// ---- Library/10_Machine/18_HMI_Handshake/OLD_DUTs/E_PullOutConveyorCommandType.TcDUT
{attribute 'qualified_only'}
{attribute 'strict'}
TYPE
    E_PullOutConveyorCommandType :
    (
		SideA_FeedIn := 1, // Pull out conveyor A-side feed in box.
		SideB_FeedIn , // Pull out conveyor B-Side feed in box.
		Both_FeedIn, // Pull out conveyor both side feed in box.
		SideA_FeedOut, // Pull out conveyor A-side feed out box.
		SideB_FeedOut, // Pull out conveyor B-Side feed out box.
		Both_FeedOut, // Pull out conveyor both side feed out box.
        MoveForward, // Pull out conveyor motor move forward.
        MoveBackward, // Pull out conveyor motor move backward.
		SlideA_FeedOut_Ext, // Pullout Conveyor A-side feed out box, fast flow(Design by Johnson)
		SlideB_FeedOut_Ext, // Pullout Conveyor B-Side feed out box, fast flow(Design by Johnson)
		SlideA_FeedIn_Ext, // Pullout Conveyor A-side feed in box, fast flow(Design by Johnson)
		SlideB_FeedIn_Ext // Pullout Conveyor B-side feed in box, fast flow(Design by Johnson)
    );
END_TYPE

// ---- Library/10_Machine/18_HMI_Handshake/OLD_DUTs/E_PullOutConveyorState.TcDUT
{attribute 'qualified_only'}
{attribute 'strict'}
TYPE E_PullOutConveyorState :
(
	idle := 0,
	AutoMode,
	Free
);
END_TYPE

// ---- Library/10_Machine/18_HMI_Handshake/OLD_DUTs/E_RackState.TcDUT
{attribute 'qualified_only'}
{attribute 'strict'}
TYPE E_RackState :
(
	idle := 0,
	AddBoxes,
	ManualCtrl,
	FeedBox,
	Free,
	TransitingFeedBox,
	TransitingFree
);
END_TYPE

// ---- Library/10_Machine/18_HMI_Handshake/OLD_DUTs/E_ReloadRoundBelt_PickupArea.TcDUT
{attribute 'qualified_only'}
{attribute 'strict'}
TYPE
    E_ReloadRoundBelt_PickupArea :
    (
        Undefined := 0,
        WareHouseA := 1,
        WareHouseB := 2
        )UINT;
END_TYPE

// ---- Library/10_Machine/18_HMI_Handshake/OLD_DUTs/E_ReloadRoundBelt_PlaceAddress.TcDUT
{attribute 'qualified_only'}
{attribute 'strict'}
TYPE E_ReloadRoundBelt_PlaceAddress :
(
	Undefined := 0,
	A1,
	A2,
	A3,
	A4
);
END_TYPE

// ---- Library/10_Machine/18_HMI_Handshake/OLD_DUTs/E_ReloadRoundBelt_PlaceArea.TcDUT
{attribute 'qualified_only'}
{attribute 'strict'}
TYPE E_ReloadRoundBelt_PlaceArea :
(
	Undefined := 0,
	RoundBelt
)UINT;
END_TYPE

// ---- Library/10_Machine/18_HMI_Handshake/OLD_DUTs/E_RobotArea.TcDUT
{attribute 'qualified_only'}
{attribute 'strict'}
(* This enum is use to define Fanuc robot target position in the StorageArea,
In the StorageArea, areas excluding the Warehouse.
*)
TYPE
    E_RobotArea :
    (
        Undefined := 0,
        // 圓帶,B區
        RoundBelt := 1,
        // 緩衝區,C區
        BufferArea := 2,
        // 補料軌道,D區
        TransmitCV := 3,
//        // 簡易配針區,E區
//        SimpleAllocate := 4,
        // 入出料軌道,F區 (倉儲區軌道)
        InOutConveyor := 5,
//        // 倉儲預備區,G區
//        WareHouseA_Buffer := 6,
        // 回拔輸送帶,H區
        PullOutConveyor := 7,
        // 小手臂左 (操作面)
        ShippingRobotLeft := 8,
        // 小手臂右 (操作面)
        ShippingRobotRight := 9,
		// Shipping Store,K
		TransmitCV_End :=10,
		// Shipping Buffer , K
		ShippingBufferArea := 11,
		// 小手臂CCD Pos
		ShippingCCDPos	:= 12,
		// 小手臂 拔針排空盒
		ShippingFeedOutEmptyBox := 13
    );
END_TYPE

// ---- Library/10_Machine/18_HMI_Handshake/OLD_DUTs/E_RobotClamp.TcDUT
{attribute 'qualified_only'}
{attribute 'strict'}
TYPE E_RobotClamp :
(
	ClampA := 1,
	ClampB
);
END_TYPE

// ---- Library/10_Machine/18_HMI_Handshake/OLD_DUTs/E_RoundBeltStation.TcDUT
{attribute 'qualified_only'}
TYPE E_RoundBeltStation :
(
	Undefined := 0,
	Station01,
	Station02,
	Station03,
	Station04,
	Station05,
	Station06,
	Station07,
	Station08,
	Station09,
	Station10,
	Station11,
	Station12,
	Station13,
	Station14,
	Station15,
	Station16,
	Station17,
	Station18,
	Station19,
	Station20,
	Station21,
	Station22,
	Station23,
	Station24,
	Station25,
	Station26,
	Station27,
	Station28,
	Station29,
	Station30,
	Station31,
	Station32,
	Station33,
	Station34,
	Station35,
	Station36,
	Station37,
	Station38,
	Station39,
	Station40
)UINT;
END_TYPE

// ---- Library/10_Machine/18_HMI_Handshake/OLD_DUTs/E_SimpleAllocateTable.TcDUT
{attribute 'qualified_only'}
{attribute 'strict'}
TYPE E_SimpleAllocateTable :
(
    Box1 :=1,
    Box2,
    Box3,
    Box4
);
END_TYPE

// ---- Library/10_Machine/18_HMI_Handshake/OLD_DUTs/E_WareHouse.TcDUT
TYPE E_WareHouse :
(
	None := 0,
	WareHouseA := 1,
	WareHouseB := 2
);
END_TYPE

// ---- Library/10_Machine/18_HMI_Handshake/OLD_DUTs/E_WareHouseLayer.TcDUT
TYPE E_WareHouseLayer :
(
	Undefine := 0,
	Layer01 := 1,
	Layer02,
	Layer03,
	Layer04,
	Layer05,
	Layer06,
	Layer07,
	Layer08,
	Layer09,
	Layer10
);
END_TYPE

// ---- Library/10_Machine/18_HMI_Handshake/OLD_DUTs/E_WareHouseSlide.TcDUT
TYPE
    E_WareHouseSlide :
    (
        Undefine := 0,
        Slide01 := 1,
        Slide02,
        Slide03,
        Slide04,
        Slide05,
        Slide06,
        Slide07,
        Slide08,
        Slide09,
        Slide10,
        Slide11,
        Slide12,
        Slide13,
        Slide14,
        Slide15,
        Slide16,
        Slide17,
        Slide18,
        Slide19,
        Slide20
    );
END_TYPE

// ---- Library/10_Machine/18_HMI_Handshake/OLD_DUTs/stPositionCommand.TcDUT
TYPE
    stPositionCommand :
    STRUCT
        Xaxis_Pos : LREAL; // Robot X-axis position command
        Yaxis_Pos : LREAL; // Robot Y-axis position command
        Raxis_Pos : LREAL; // Robot R-axis Position command
    END_STRUCT
END_TYPE

// ---- Library/10_Machine/18_HMI_Handshake/OLD_DUTs/st_ads_AllocateMoveStructure.TcDUT
TYPE
    st_ads_AllocateMoveStructure :
    STRUCT
        //手臂夾爪 ex 0=>A爪 1=>B爪 and so on...	
        Clip         : LREAL;
        Frombox      : LREAL;
        Tobox        : LREAL;
        FromPosition : LREAL;
        ToPosition   : LREAL;
        HandShake    : st_HandshakeBase;
    END_STRUCT
END_TYPE

// ---- Library/10_Machine/18_HMI_Handshake/OLD_DUTs/st_ads_MachineReset.TcDUT
TYPE st_ads_MachineReset :
    STRUCT
        //清除各分區除了伺服軸外的所有動件(氣壓缸、馬達)的邏輯層錯誤
        ResetStorage    :BOOL;
        ResetAllocation :BOOL;
        ResetFGA        :BOOL;
        AllReset        :BOOL;// Machine reset signal, True: machine try to clear alarm and reset method 
    END_STRUCT
END_TYPE

// ---- Library/10_Machine/18_HMI_Handshake/OLD_DUTs/st_ads_OneAxisMoveWithoutPosition.TcDUT
TYPE st_ads_OneAxisMoveWithoutPosition :
STRUCT
	//Excute:BOOL;
	//Done:BOOL;
	//Busy  : BOOL;
	//Occupied : BOOL;
	
	HandShake					: st_HandshakeBase;
END_STRUCT
END_TYPE

// ---- Library/10_Machine/18_HMI_Handshake/OLD_DUTs/st_ads_OneAxisMoveWithPosition.TcDUT
TYPE st_ads_OneAxisMoveWithPosition :
STRUCT
	Clip:LREAL;
	Position:LREAL; 
	
	HandShake					: st_HandshakeBase;
END_STRUCT
END_TYPE

// ---- Library/10_Machine/18_HMI_Handshake/OLD_DUTs/st_ads_OutRobtToPlateMove.TcDUT
TYPE st_ads_OutRobtToPlateMove :
STRUCT
	//軌道 散針軌道 or 同尺寸軌道
Slide :LREAL;
Clip:LREAL;
//鐵盤位置
PlatePosition :LREAL;
//Excute :bool;
//Done    :BOOL;
HandShake					: st_HandshakeBase;
END_STRUCT
END_TYPE

// ---- Library/10_Machine/18_HMI_Handshake/OLD_DUTs/st_ads_RobotToAllocateMove.TcDUT
TYPE
    st_ads_RobotToAllocateMove :
    STRUCT
        //圓帶位置
        AllocatePosition : LREAL;
        //手臂夾爪 ex 0=>A爪 1=>B爪
        RobotClip : LREAL;
        //倉儲區域 ex>A,B
        Area : LREAL;
        //倉儲層
        WarehouseLayer : LREAL;
        //倉儲道
        WarehouseOrbit : LREAL;
        // :BOOL;
        //Done :BOOL;
        HandShake : st_HandshakeBase;
    END_STRUCT
END_TYPE

// ---- Library/10_Machine/18_HMI_Handshake/OLD_DUTs/ST_Alarm_Tmax.TcDUT
TYPE ST_Alarm_Tmax :
STRUCT
		Trigger		:BOOL; //	Alarm trigger point
		ID			: UDINT; //	Alarm ID
		Value		: DINT; //	Alarm Value
		Message		: T_MaxString; //	Alarm Message
		Category	: DINT; //	Alarm Category
		DateTime	: ARRAY[0..6] OF DINT;
		ackDateTime : ARRAY[0..6] OF DINT;
END_STRUCT
END_TYPE

// ---- Library/10_Machine/18_HMI_Handshake/OLD_DUTs/st_AllocateCircleMoveStructure.TcDUT
TYPE st_AllocateCircleMoveStructure :
STRUCT
	Latch : LREAL;
	Position :LREAL;
//	Excute	:BOOL;
//	Done	 :BOOL;
//	Busy  : BOOL;
//	Occupied : BOOL;	
	HandShake					: st_HandshakeBase;
END_STRUCT
END_TYPE

// ---- Library/10_Machine/18_HMI_Handshake/OLD_DUTs/st_AllocateRobotNeedlingMove.TcDUT
TYPE st_AllocateRobotNeedlingMove :
STRUCT
	Command 	: ST_CommandBasic;
	Status 		: ST_StatusBasic;
	MovingInfo	: ST_AllocateRobotNeedlingMoveInfo;
END_STRUCT
END_TYPE

// ---- Library/10_Machine/18_HMI_Handshake/OLD_DUTs/ST_AllocateRobotNeedlingMoveInfo.TcDUT
TYPE ST_AllocateRobotNeedlingMoveInfo :
STRUCT
	NeedleLocation		: INT;	//針位，0~49
	Box					: UINT;	//盒位，0~3
	Clip				: INT;	//使用夾爪，0~3
	Area				: STRING; // Q : 圓帶 T :轉盤

END_STRUCT
END_TYPE

// ---- Library/10_Machine/18_HMI_Handshake/OLD_DUTs/st_AllocatingNeedleInfo.TcDUT
TYPE st_AllocatingNeedleInfo :
STRUCT
	NeedleLocation		: INT;	//針位，0~49
	Box					: UINT;	//盒位，0~3
	Clip				: INT;	//使用夾爪，0~3(可新增到5)
	Station				: UINT;	//圓帶站點 ，(放針時無效) 1..40
	CycleStart			: BOOL;	//取到此針後執行放針，討論放針做為作動依據
END_STRUCT
END_TYPE

// ---- Library/10_Machine/18_HMI_Handshake/OLD_DUTs/ST_AllocationJobBatchMode.TcDUT
TYPE ST_AllocationJobBatchMode :
STRUCT
	AllocationInfo		: ARRAY[0..49] OF ST_AllocationJobBatchModeInfo; //Max 50 allocation jobs once
	HandShake			: st_HandshakeBase;
	NrOfAllocationJob	: UINT; // How many jobs this batch , Max :50
	Pause				: BOOL;
	WorkedID			:  ARRAY[0..49] OF INT;	 // feedback which job was done , start in -1 means not finishing any job yet

END_STRUCT
END_TYPE

// ---- Library/10_Machine/18_HMI_Handshake/OLD_DUTs/ST_AllocationJobBatchModeInfo.TcDUT
TYPE ST_AllocationJobBatchModeInfo :
STRUCT
	PickingNeedleInfo			: ARRAY[0..3] OF st_AllocatingNeedleInfo;	//取針資料
	PlacingNeedleInfo			: ARRAY[0..3] OF st_AllocatingNeedleInfo;	//放針資料
	FastMode					: BOOL;
	SyncMode					: BOOL;
	ID							: INT;   // -1 means null , do not use
END_STRUCT
END_TYPE

// ---- Library/10_Machine/18_HMI_Handshake/OLD_DUTs/ST_AllocationJobBatchMode_1.TcDUT
TYPE ST_AllocationJobBatchMode_1 :
STRUCT
	AllocationInfo		: ARRAY[0..49] OF ST_AllocationJobBatchModeInfo; //Max 50 allocation jobs once
	HandShake			: st_HandshakeBase;
	NrOfAllocationJob	: UINT; // How many jobs this batch , Max :50
	Pause				: BOOL;
	WorkedID			:  ARRAY[0..49] OF INT;	 // feedback which job was done , start in -1 means not finishing any job yet

END_STRUCT
END_TYPE

// ---- Library/10_Machine/18_HMI_Handshake/OLD_DUTs/ST_AutoAddsBoxes.TcDUT
TYPE ST_AutoAddsBoxes :
STRUCT
	Command	: ST_AutoAddsBoxesCommand;
	Status	: ST_AutoAddsBoxesStatus;
END_STRUCT
END_TYPE

// ---- Library/10_Machine/18_HMI_Handshake/OLD_DUTs/ST_AutoAddsBoxesCommand.TcDUT
TYPE ST_AutoAddsBoxesCommand EXTENDS ST_CommandBasic :
STRUCT
END_STRUCT
END_TYPE

// ---- Library/10_Machine/18_HMI_Handshake/OLD_DUTs/ST_AutoAddsBoxesStatus.TcDUT
TYPE ST_AutoAddsBoxesStatus EXTENDS ST_StatusBasic :
STRUCT
	InterventionRequest	 : BOOL;
	FeedingBoxes		 :BOOL;
END_STRUCT
END_TYPE

// ---- Library/10_Machine/18_HMI_Handshake/OLD_DUTs/st_AutoMode_AllocatingJob.TcDUT
TYPE st_AutoMode_AllocatingJob :
STRUCT
	PickingNeedleInfo			: Array[0..3] OF st_AllocatingNeedleInfo;	//取針資料
	PlacingNeedleInfo			: ARRAY[0..3] OF st_AllocatingNeedleInfo;	//放針資料
	FastMode					: BOOL;
	SyncMode					: BOOL;
	HandShake					: st_HandshakeBase;
END_STRUCT
END_TYPE

// ---- Library/10_Machine/18_HMI_Handshake/OLD_DUTs/st_AutoMode_AllocatingJob_1.TcDUT
TYPE st_AutoMode_AllocatingJob_1 :
STRUCT
	PickingNeedleInfo			: Array[0..3] OF st_AllocatingNeedleInfo;	//取針資料
	PlacingNeedleInfo			: ARRAY[0..3] OF st_AllocatingNeedleInfo;	//放針資料
	FastMode					: BOOL;
	SyncMode					: BOOL;
	HandShake					: st_HandshakeBase;
END_STRUCT
END_TYPE

// ---- Library/10_Machine/18_HMI_Handshake/OLD_DUTs/st_AutoMode_ClampingBoxesJob.TcDUT
TYPE st_AutoMode_ClampingBoxesJob :
STRUCT
	ClampingInfo			: st_ClampingBoxesInfo;
	HandShake				: st_HandshakeBase;
END_STRUCT
END_TYPE

// ---- Library/10_Machine/18_HMI_Handshake/OLD_DUTs/st_AutoMode_ClampingToPlate.TcDUT
TYPE st_AutoMode_ClampingToPlate :
STRUCT
	ClampingInfo			: st_ClampingBoxesInfo;
	ClipAFrom				: INT; //0: 配好輸送帶。1: 同尺吋輸送帶
	ClipBFrom				: INT; //0: 配好輸送帶。1: 同尺吋輸送帶
	HandShake				: st_HandshakeBase;
END_STRUCT
END_TYPE

// ---- Library/10_Machine/18_HMI_Handshake/OLD_DUTs/ST_AutoMode_DetectDiameter.TcDUT
TYPE ST_AutoMode_DetectDiameter :
STRUCT
	Command: ST_DetectDiameterCommand;
	Status: ST_DetectDiameterStatus;
	DetectDiameterInfo:ST_DetectDiameterInfo;
END_STRUCT
END_TYPE

// ---- Library/10_Machine/18_HMI_Handshake/OLD_DUTs/ST_AutoMode_FeedInEmptyBox.TcDUT
TYPE ST_AutoMode_FeedInEmptyBox :
STRUCT
	Command : ST_FeedInEmptyBox_Ctrl;
	Status : ST_FeedInEmptyBox_Status;
	Info : ST_FeedInEmptyBox_Info;
	AClampMoveDone	: BOOL;		//edited by Gamin 2025/11/24
	BClampMoveDone	: BOOL;
END_STRUCT
END_TYPE

// ---- Library/10_Machine/18_HMI_Handshake/OLD_DUTs/ST_AutoMode_ReloadRoundBeltBox.TcDUT
TYPE ST_AutoMode_ReloadRoundBeltBox :
STRUCT
	Command : ST_ReloadRoundBelt_Ctrl;
	Status : ST_ReloadRoundBelt_Status;
	Info : ST_ReloadRoundBeltBox_Info;
	AClampMoveDone	: BOOL;
	BClampMoveDone	: BOOL;
END_STRUCT
END_TYPE

// ---- Library/10_Machine/18_HMI_Handshake/OLD_DUTs/ST_AutoMode_RobotRegionMove.TcDUT
TYPE ST_AutoMode_RobotRegionMove :
STRUCT
	Command 	: ST_CommandBasic;
	Status 		: ST_StatusBasic;
	Info 		: ST_RobotRegionMove_Info;
END_STRUCT
END_TYPE

// ---- Library/10_Machine/18_HMI_Handshake/OLD_DUTs/ST_AutoMode_ShippingLeftSideTransCVFeedBack.TcDUT
TYPE ST_AutoMode_ShippingLeftSideTransCVFeedBack :
STRUCT
	TransCV_IntargetPosition : BOOL;
END_STRUCT
END_TYPE

// ---- Library/10_Machine/18_HMI_Handshake/OLD_DUTs/ST_AutoMode_ShippingLeftSideTransCVInfo.TcDUT
TYPE ST_AutoMode_ShippingLeftSideTransCVInfo :
STRUCT
	ShippingTransCVRequest : BOOL;
END_STRUCT
END_TYPE

// ---- Library/10_Machine/18_HMI_Handshake/OLD_DUTs/ST_AutoMode_ShippingRightSideTransCV.TcDUT
TYPE ST_AutoMode_ShippingRightSideTransCV :
STRUCT
	Command : ST_CommandBasic;
	Status	: ST_StatusBasic;
	ShippingTransCVRequest_RightSide : BOOL;		//C# to PLC
END_STRUCT
END_TYPE

// ---- Library/10_Machine/18_HMI_Handshake/OLD_DUTs/ST_AutoMode_SimpleAllocateHandShake.TcDUT
TYPE ST_AutoMode_SimpleAllocateHandShake :
    STRUCT
        Command            :ST_SimpleAllocateCommand; // Commands about simple allocate function
        Status             :ST_SimpleAllocateStatus; // Status about simple allocate function
        SimpleAllocateInfo :ST_SimpleAllocateInfo; // Parameters about simple allocate function
    END_STRUCT
END_TYPE

// ---- Library/10_Machine/18_HMI_Handshake/OLD_DUTs/st_AutoMode_SingleStepWithInterventionRequest.TcDUT
TYPE st_AutoMode_SingleStepWithInterventionRequest :
STRUCT
	InterventionRequest	 : BOOL;
	HandShake		: st_HandshakeBase;
END_STRUCT
END_TYPE

// ---- Library/10_Machine/18_HMI_Handshake/OLD_DUTs/ST_AutoMode_TransCVCamera.TcDUT
TYPE ST_AutoMode_TransCVCamera :
STRUCT
	Command :ST_CommandBasic;
	Status	:ST_StatusBasic;
	UseBoxCamera	:BOOL;
	BoxCameraDone	:BOOL;
END_STRUCT
END_TYPE

// ---- Library/10_Machine/18_HMI_Handshake/OLD_DUTs/ST_AutoMode_WareHouseInnerPickToRoundBelt.TcDUT
// 倉儲內取放圓帶 — 自動模式包裝結構 (單筆)
// 提供 Command/Status 握手 + 流程資訊 + 動作紀錄陣列
// C# 透過 ADS 讀取 FeedBack=TRUE 後批次讀取 ActionRecords
TYPE ST_AutoMode_WareHouseInnerPickToRoundBelt :
STRUCT
	Command			: ST_CommandBasic;		// Execute / Abort / Reset 控制命令
	Status			: ST_StatusBasic;		// Busy / Done / Error / Status 狀態回報
	Info			: ST_WareHouseInnerPickFlowInfo;	// 單筆流程資訊 (A/B爪設定+深度)
	ActionRecords	: ARRAY[0..39] OF ST_ClampActionRecord;	// 倉儲取放動作紀錄
	ActionIndex		: INT;					// 已記錄筆數
	FeedBack		: BOOL;					// PLC → C#: 陣列可讀取
	ReadComplete	: BOOL;					// C# → PLC: 讀取完成確認
END_STRUCT
END_TYPE

// ---- Library/10_Machine/18_HMI_Handshake/OLD_DUTs/E_ShippingPlateIndex.TcDUT
{attribute 'qualified_only'}
{attribute 'strict'}
(* enum 值 = 手臂 Position，PLC 內可直接 INT(PlateIndex) 送 robot *)
TYPE E_ShippingPlateIndex :
(
	Plate1	:= 1,
	Plate2	:= 2,
	Plate3	:= 3,
	Plate4	:= 4
);
END_TYPE

// ---- Library/10_Machine/18_HMI_Handshake/OLD_DUTs/E_ShippingPlateSide.TcDUT
{attribute 'qualified_only'}
{attribute 'strict'}
TYPE E_ShippingPlateSide :
(
	Left	:= 0,
	Right	:= 1
);
END_TYPE

// ---- Library/10_Machine/18_HMI_Handshake/OLD_DUTs/ST_ShippingPlateToConveyor.TcDUT
TYPE ST_ShippingPlateToConveyor :
STRUCT
	Command			: ST_CommandBasic;
	Status			: ST_StatusBasic;

	// C# >> PLC (上位決定)
	Side			: E_ShippingPlateSide;		// Left=0 / Right=1
	PlateIndex		: E_ShippingPlateIndex;		// Plate1..Plate4
	ReadComplete	: BOOL;						// 上位讀完 PlateHasBox 後回 TRUE

	// PLC >> C#
	PlateHasBox		: BOOL;		// 該次掃描有沒有盒子 (Robot._DI13.9)
	FeedBack		: BOOL;		// 掃完待讀,等 ReadComplete
END_STRUCT
END_TYPE

// ---- Library/10_Machine/18_HMI_Handshake/OLD_DUTs/ST_AutoPullOutConveyor.TcDUT
TYPE ST_AutoPullOutConveyor :
STRUCT
	PullOutConveyorInfo : ST_PullOutConveyorInfo;
	Command :ST_AutoPullOutConveyorCommand;
	Status : ST_AutoPullOutConveyorSatus;
END_STRUCT
END_TYPE

// ---- Library/10_Machine/18_HMI_Handshake/OLD_DUTs/ST_AutoPullOutConveyorCommand.TcDUT
TYPE ST_AutoPullOutConveyorCommand EXTENDS ST_CommandBasic :
STRUCT
END_STRUCT
END_TYPE

// ---- Library/10_Machine/18_HMI_Handshake/OLD_DUTs/ST_AutoPullOutConveyorSatus.TcDUT
TYPE ST_AutoPullOutConveyorSatus EXTENDS ST_StatusBasic :
STRUCT
END_STRUCT
END_TYPE

// ---- Library/10_Machine/18_HMI_Handshake/OLD_DUTs/ST_AutoServoPara.TcDUT
TYPE ST_AutoServoPara :
    STRUCT
        Position :LREAL;
        Velocity :LREAL;
        Distance :LREAL;
        ACC      :LREAL;
        DEC      :LREAL;
        Jerk     :LREAL;
    END_STRUCT
END_TYPE

// ---- Library/10_Machine/18_HMI_Handshake/OLD_DUTs/st_AutoSixAxisAbsMoveParameter.TcDUT
TYPE st_AutoSixAxisAbsMoveParameter :
STRUCT
	A_Area:LREAL;
	B_Area:LREAL;
	A_Position:LREAL;
	B_Position:LREAL;
	A_Get:BOOL;
	B_Get:BOOL;
	AClampMoveDone	: BOOL;
	BClampMoveDone	: BOOL;
	(*Excute:BOOL;
	Done  :BOOL;
	Busy  : BOOL;
	Occupied : BOOL;
	Error : BOOL;	*)
	HandShake				: st_HandshakeBase;
END_STRUCT
END_TYPE

// ---- Library/10_Machine/18_HMI_Handshake/OLD_DUTs/st_AutoSixAxisWarehouseParameter.TcDUT
TYPE st_AutoSixAxisWarehouseParameter :
STRUCT
	Warehouse_A	:	BOOL; //58ON = TRUE, 59ON = FALSE
	Warehouse_B	:	BOOL; //74ON = TRUE, 75ON = FALSE
	Layer_A 	: 	LREAL;
	Layer_B 	:	LREAL;
	Slide_A 	:	LREAL;
	Slide_B 	:	LREAL;	
	Get_A		:	BOOL;
	Get_B		:	BOOL;
	AClampMoveDone	: BOOL;
	BClampMoveDone	: BOOL;
	(*Excute		:	BOOL;
	Done  		:	BOOL;
	Busy  		:	BOOL;
	Occupied 	:	BOOL;
	Error		:	BOOL;
	Reset		:	BOOL;*)
	HandShake				: st_HandshakeBase;
END_STRUCT
END_TYPE

// ---- Library/10_Machine/18_HMI_Handshake/OLD_DUTs/st_AutoSperate.TcDUT
TYPE st_AutoSperate :
STRUCT
Clips  		: ARRAY[0..4] OF BOOL; // Working Clips this round
Position 	: INT;				   // Position index 0~7
Row 		: INT;				   // Row of Needle 0~4
HandShake	: st_HandshakeBase;	   // Handshake
END_STRUCT
END_TYPE

// ---- Library/10_Machine/18_HMI_Handshake/OLD_DUTs/ST_Auto_LowerFeedInConveyor.TcDUT
TYPE ST_Auto_LowerFeedInConveyor :
STRUCT
	Command :ST_Auto_LowerFeedInConveyorCommand;
	Status	:ST_Auto_LowerFeedInConveyorStatus;
END_STRUCT
END_TYPE

// ---- Library/10_Machine/18_HMI_Handshake/OLD_DUTs/ST_Auto_LowerFeedInConveyorCommand.TcDUT
TYPE ST_Auto_LowerFeedInConveyorCommand EXTENDS ST_CommandBasic :
STRUCT
END_STRUCT
END_TYPE

// ---- Library/10_Machine/18_HMI_Handshake/OLD_DUTs/ST_Auto_LowerFeedInConveyorStatus.TcDUT
TYPE ST_Auto_LowerFeedInConveyorStatus EXTENDS ST_StatusBasic :
STRUCT
END_STRUCT
END_TYPE

// ---- Library/10_Machine/18_HMI_Handshake/OLD_DUTs/ST_Auto_UpperFeedInConveyor.TcDUT
TYPE ST_Auto_UpperFeedInConveyor :
STRUCT
	Command		: ST_Auto_UpperFeedInConveyorCommand;
	Status		: ST_Auto_UpperFeedInConveyorStatus;	
	Info		: ST_Auto_UpperFeedInConveyorInfo;
	FeedBack    : ST_Auto_UpperFeedInConveyorFeedback;	
	
END_STRUCT
END_TYPE

// ---- Library/10_Machine/18_HMI_Handshake/OLD_DUTs/ST_Auto_UpperFeedInConveyorCommand.TcDUT
TYPE ST_Auto_UpperFeedInConveyorCommand EXTENDS ST_CommandBasic :
STRUCT
END_STRUCT
END_TYPE

// ---- Library/10_Machine/18_HMI_Handshake/OLD_DUTs/ST_Auto_UpperFeedInConveyorFeedback.TcDUT
TYPE ST_Auto_UpperFeedInConveyorFeedback :
STRUCT
	FirstBoxCamera : BOOL;
	SecondBoxCamera : BOOL;	
	FirstBoxCameraDiameter : BOOL;
	SecondBoxCameraDiameter : BOOL;
	ActualNrOfBox			:INT;
	InterventionRequest	 : BOOL;
END_STRUCT
END_TYPE

// ---- Library/10_Machine/18_HMI_Handshake/OLD_DUTs/ST_Auto_UpperFeedInConveyorInfo.TcDUT
TYPE ST_Auto_UpperFeedInConveyorInfo :
STRUCT
	NrOfBox		: INT ; // 1 or 2
	FirstBoxCameraDone 				: BOOL;
	SecondBoxCameraDone 			: BOOL;
	
	FirstBoxCameraDiameterRequest 	: BOOL;
	SecondBoxCameraDiameterRequest 	: BOOL;
	
	FirstBoxCameraDiameterDone 		: BOOL;
	SecondBoxCameraDiameterDone 	: BOOL;
	
	FeedAirblowTime 				:TIME;
END_STRUCT
END_TYPE

// ---- Library/10_Machine/18_HMI_Handshake/OLD_DUTs/ST_Auto_UpperFeedInConveyorStatus.TcDUT
TYPE ST_Auto_UpperFeedInConveyorStatus EXTENDS ST_StatusBasic :
STRUCT
END_STRUCT
END_TYPE

// ---- Library/10_Machine/18_HMI_Handshake/OLD_DUTs/st_AxisControl.TcDUT
TYPE st_AxisControl :
STRUCT
	Error	  : BOOL;
	ResetAxis : BOOL;
END_STRUCT
END_TYPE

// ---- Library/10_Machine/18_HMI_Handshake/OLD_DUTs/ST_BuzzCtrl.TcDUT
TYPE ST_BuzzCtrl :
STRUCT
	Command : ST_CommandBasic;
	Status	: ST_StatusBasic;
	BuzzTime	: LREAL;
END_STRUCT
END_TYPE

// ---- Library/10_Machine/18_HMI_Handshake/OLD_DUTs/ST_ClampActionRecord.TcDUT
// 倉儲取放動作紀錄 — 每次從倉儲取盒或放回倉儲時記錄一筆
// 由 FB_WareHouseInnerPickToRoundBelt 在動作完成時寫入
// C# 透過 ADS 讀取 FeedBack=TRUE 後批次讀取整個陣列
TYPE ST_ClampActionRecord :
STRUCT
	WareHouse	: INT;		// 倉別 (E_WareHouse 對應值)
	Layer		: INT;		// 層 (E_WAREHOUSELAYER 對應值)
	Slide		: INT;		// 軌道 (E_WAREHOUSESLIDE 對應值)
	Clamp		: INT;		// 0 = A爪, 1 = B爪
	IsPick		: BOOL;		// TRUE = 取盒 (從倉儲取出), FALSE = 放盒 (放回倉儲)
END_STRUCT
END_TYPE

// ---- Library/10_Machine/18_HMI_Handshake/OLD_DUTs/st_ClampingBoxesInfo.TcDUT
TYPE st_ClampingBoxesInfo :
STRUCT
	NrOfBoxes		: INT;	// 1,2
	TargetOfClipA	: INT;	// 0 : R1, 1: R2 or To plate index
	TargetOfClipB	: INT;	// 0 : R1, 1: R2 or To plate index
	UseClibA		: BOOL;	//Clip A only work if True
	UseClibB		: BOOL;	//Clip B only work if True
END_STRUCT
END_TYPE

// ---- Library/10_Machine/18_HMI_Handshake/OLD_DUTs/ST_ClampSetting.TcDUT
TYPE
    ST_ClampSetting :
    STRUCT
        Behavior         : E_ClampWork;
        WareHouseSetting : ST_WareHouseCoordinates;
		PullOutConveyorSetting : E_PullOutConveyorAddress;
        PickUpArea : E_FeedInEmptyBox_PickUpArea; // Set the position where are the Fanuc robot going to pickup box.
        PlaceArea  : E_FeedInEmptyBox_PlaceArea; // Set the position where are the Fanuc robot going to place box.
    END_STRUCT
END_TYPE

// ---- Library/10_Machine/18_HMI_Handshake/OLD_DUTs/ST_ClampSetting_FeedInToWareHouse.TcDUT
TYPE
    ST_ClampSetting_FeedInToWareHouse :
    STRUCT
        Behavior         : E_ClampWork;                          // Work or NoWork
        RoundBeltSetting : ST_RoundBeltCoordinates;              // RoundBelt station and carrier position (A2/A3) for pickup
        WareHouseSetting : ST_WareHouseCoordinates;              // WareHouse layer and slide for placement
        PlaceArea        : E_FeedInToWareHouse_PlaceArea;        // Target warehouse (WareHouseA or WareHouseB)
    END_STRUCT
END_TYPE

// ---- Library/10_Machine/18_HMI_Handshake/OLD_DUTs/ST_ClampSetting_ReloadRoundBelt.TcDUT
TYPE
    ST_ClampSetting_ReloadRoundBelt :
    STRUCT
        Behavior         : E_ClampWork;
        WareHouseSetting : ST_WareHouseCoordinates;
		RoundBeltSetting : ST_RoundBeltCoordinates; // Set Clamp to which pos work
        PickUpArea       : E_ReloadRoundBelt_PickupArea; // Set the position where are the Fanuc robot going to pickup box.
        PlaceArea        : E_ReloadRoundBelt_PlaceArea := E_ReloadRoundBelt_PlaceArea.RoundBelt; // Set the position where are the Fanuc robot going to place box.
    END_STRUCT
END_TYPE

// ---- Library/10_Machine/18_HMI_Handshake/OLD_DUTs/ST_CommandBasic.TcDUT
TYPE ST_CommandBasic :
    STRUCT
        Execute :BOOL; // TRUE : Process start
        Abort   :BOOL; // TRUE : Process abort
        Reset   :BOOL; // TRUE : Process reset
    END_STRUCT
END_TYPE

// ---- Library/10_Machine/18_HMI_Handshake/OLD_DUTs/ST_DetectDiameterCommand.TcDUT
TYPE ST_DetectDiameterCommand EXTENDS ST_CommandBasic :
STRUCT
	GetPhotoCompleted : BOOL;
END_STRUCT
END_TYPE

// ---- Library/10_Machine/18_HMI_Handshake/OLD_DUTs/ST_DetectDiameterInfo.TcDUT
TYPE ST_DetectDiameterInfo :
STRUCT
	ClampA_Used : BOOL;
	ClampB_Used : BOOL;
END_STRUCT
END_TYPE

// ---- Library/10_Machine/18_HMI_Handshake/OLD_DUTs/ST_DetectDiameterStatus.TcDUT
TYPE ST_DetectDiameterStatus EXTENDS ST_StatusBasic :
STRUCT
	AllowGetPhoto : BOOL;
END_STRUCT
END_TYPE

// ---- Library/10_Machine/18_HMI_Handshake/OLD_DUTs/ST_FanucRobotGeneralCtrl.TcDUT
TYPE ST_FanucRobotGeneralCtrl :
STRUCT
	Command : ST_FanucRobot_CSharpCommand;
	Status : ST_FanucRobot_CSharpStatus;
END_STRUCT
END_TYPE

// ---- Library/10_Machine/18_HMI_Handshake/OLD_DUTs/ST_FanucRobotReadAllOffssetDate.TcDUT
TYPE ST_FanucRobotReadAllOffssetDate :
STRUCT
	Command	: ST_ReadAllOffsetDataCommand; // Read all offset data command struct.
	Status 	: ST_ReadAllOffsetDateStatus; // Read all offset data status struct.
//	Info	: ST_ReadAllOffsetDataInfo; //Read all offset dara info struct.
END_STRUCT
END_TYPE

// ---- Library/10_Machine/18_HMI_Handshake/OLD_DUTs/ST_FanucRobotReadSingleOffsetData.TcDUT
TYPE ST_FanucRobotReadSingleOffsetData :
STRUCT
	Command : ST_ReadSingleOffsetData_Command;
	Status 	: ST_ReadSingleOffsetData_Status;
	Info	: ST_ReadSingleOffsetData_Info;
END_STRUCT
END_TYPE

// ---- Library/10_Machine/18_HMI_Handshake/OLD_DUTs/ST_FanucRobotWriteAllOffsetDate.TcDUT
TYPE ST_FanucRobotWriteAllOffsetDate :
STRUCT
	Command : ST_WriteAllOffsetData_Command;
	Status	: ST_WriteAllOffsetData_Status;
	Info	: ST_WriteAllOffsetData_Info;
END_STRUCT
END_TYPE

// ---- Library/10_Machine/18_HMI_Handshake/OLD_DUTs/ST_FanucRobotWriteSingleOffsetData.TcDUT
TYPE ST_FanucRobotWriteSingleOffsetData :
STRUCT
	Command : ST_WriteSingleOffsetData_Command;
	Status	: ST_WriteSingleOffsetData_Status;
	Info	: ST_WriteSingleOffsetData_Info;
END_STRUCT
END_TYPE

// ---- Library/10_Machine/18_HMI_Handshake/OLD_DUTs/ST_FanucRobot_CSharpCommand.TcDUT
TYPE ST_FanucRobot_CSharpCommand :
STRUCT
	RobotVelocity : INT:=5; // Set Fanuc Robot RSR1 prog velocity command. (0~100)
	ClampA_Open  : BOOL; // True: set clampA open 
	ClampA_Close : BOOL; // True: Set ClampA Close
	ClampB_Open  : BOOL; // True: Set ClampB Open
	ClampB_Close : BOOL; // True: Set ClampB Close
	ByPassClampSensor : BOOL; // True : Bypass clampA and clampB
END_STRUCT
END_TYPE

// ---- Library/10_Machine/18_HMI_Handshake/OLD_DUTs/ST_FanucRobot_CSharpStatus.TcDUT
TYPE ST_FanucRobot_CSharpStatus :
STRUCT
	ClampA_Open : BOOL; // True : ClampA is open;
	ClampB_Open : BOOL; // True : ClampB is open;
	ClampA_Sensor : BOOL; // True : ClampA sensor has detected box.
	ClampB_Sensor : BOOL; // True : ClampB sensor hase detected box.
END_STRUCT
END_TYPE

// ---- Library/10_Machine/18_HMI_Handshake/OLD_DUTs/ST_FeedInEmptyBox_Ctrl.TcDUT
TYPE
    ST_FeedInEmptyBox_Ctrl EXTENDS ST_CommandBasic :
    STRUCT
    END_STRUCT
END_TYPE

// ---- Library/10_Machine/18_HMI_Handshake/OLD_DUTs/ST_FeedInEmptyBox_Info.TcDUT
TYPE
    ST_FeedInEmptyBox_Info :
    STRUCT
		ClampA_Setting : ST_ClampSetting; // Set clampA action.
		ClampB_Setting : ST_ClampSetting; // Set clampB action.
    END_STRUCT
END_TYPE

// ---- Library/10_Machine/18_HMI_Handshake/OLD_DUTs/ST_FeedInEmptyBox_Status.TcDUT
TYPE
    ST_FeedInEmptyBox_Status EXTENDS ST_StatusBasic :
    STRUCT
		
    END_STRUCT
END_TYPE

// ---- Library/10_Machine/18_HMI_Handshake/OLD_DUTs/ST_FeedInRBActionRecord.TcDUT
// 圓帶回倉 (FeedInRB) 動作紀錄 — 每筆 batch 流程完成時記錄
// 由 FB_FeedInRoundBeltBoxToWareHouse 的 batch handshake 模式寫入
// C# 透過 ADS 讀取 FeedBack=TRUE 後讀取整個陣列
//
// 用於記錄: 從圓帶哪一站取盒 → 放到哪個目的地 (倉儲層軌 / PullOut 內外側)
TYPE ST_FeedInRBActionRecord :
STRUCT
	// === 來源 (圓帶) ===
	PickStation		: INT;		// 圓帶 station 編號 (E_RoundBeltStation 對應值, 1..40)
	PickCarrier		: INT;		// 圓帶載具位置 (E_ReloadRoundBelt_PlaceAddress, 1=A1 / 2=A2 / 3=A3 / 4=A4)

	// === 目的 ===
	DestType		: INT;		// 0 = WareHouse, 1 = PullOut
	WareHouse		: INT;		// (DestType=0 時) 倉別 (E_WareHouse 對應值, 1=A / 2=B)
	Layer			: INT;		// (DestType=0 時) 層 (E_WAREHOUSELAYER 對應值)
	Slide			: INT;		// (DestType=0 時) 軌道 (E_WAREHOUSESLIDE 對應值)
	PullOutSide		: INT;		// (DestType=1 時) 0 = Inner (I3_Slide,左) / 1 = Outer (I4_Slide,右)

	// === 共用 ===
	Clamp			: INT;		// 0 = A爪, 1 = B爪
END_STRUCT
END_TYPE

// ---- Library/10_Machine/18_HMI_Handshake/OLD_DUTs/ST_FeedInRBBatch.TcDUT
// 圓帶回倉 (FeedInRB) — 批次結構
// 最多 40 筆流程, 由上位機 (C# HMI) 透過 ADS 寫入 FlowInfo 陣列
// 每筆流程可選擇放到 倉儲 (WareHouseA/B) 或 PullOutConveyor (Inner/Outer)
//
// HandShake 控制啟動 (Execute) / 完成 (Done) / 錯誤 (Error) / 重置 (Reset)
// WorkedID 回報每筆流程完成狀態 → C# 端據此更新 SQL 紀錄
// ActionRecords 為當前單筆流程的動作紀錄, C# 透過 FeedBack 握手讀取
//
// FeedBack/ReadComplete 跨迭代握手協定:
//   PLC: 單筆完成 → FeedBack:=TRUE → 等 ReadComplete=TRUE → 清 FeedBack → 進下一筆
//   C#:  看到 FeedBack=TRUE → 讀 ActionRecords → 寫 ReadComplete=TRUE → 等 FeedBack=FALSE → 清 ReadComplete
TYPE ST_FeedInRBBatch :
STRUCT
	FlowInfo		: ARRAY[0..39] OF ST_FeedInRBFlowInfo;		// 流程陣列, 最多 40 筆
	HandShake		: st_HandshakeBase;		// Execute/Done/Busy/Error/Reset 握手信號
	NrOfFlow		: UINT;					// 本次批次有效流程數量 (0..40)
	Pause			: BOOL;					// TRUE = 暫停批次執行 (完成當前流程後在邊界凍結)
	WorkedID		: ARRAY[0..39] OF INT;	// 完成回報: -1 = 未完成, 其餘 = 已完成的流程 ID

	// === 內層 per-iteration handshake ===
	ActionRecords	: ARRAY[0..39] OF ST_FeedInRBActionRecord;	// 當前流程的動作紀錄
	ActionIndex		: INT;		// 已記錄筆數
	FeedBack		: BOOL;		// PLC → C#: 陣列可讀取
	ReadComplete	: BOOL;		// C# → PLC: 讀取完成確認
END_STRUCT
END_TYPE

// ---- Library/10_Machine/18_HMI_Handshake/OLD_DUTs/ST_FeedInRBFlowInfo.TcDUT
// 圓帶回倉 (FeedInRB) — 單筆流程資訊
// 定義 A/B 爪各自的圓帶來源 + 目的地 (倉儲 or PullOut)
// 由上位機 (C# HMI) 透過 ADS 寫入,PLC 端根據此結構執行取放動作
//
// 跟 ST_ClampSetting_FeedInToWareHouse 共用, 但 PlaceArea 已擴充支援 PullOutInner / PullOutOuter
// 當 PlaceArea = WareHouseA/B → 使用 WareHouseSetting (Layer/Slide)
// 當 PlaceArea = PullOutInner → 對應 PullOutConveyor I3_Slide (左, 1)
// 當 PlaceArea = PullOutOuter → 對應 PullOutConveyor I4_Slide (右, 2)
TYPE ST_FeedInRBFlowInfo :
STRUCT
	ID				: INT := -1;	// 流程 ID, -1 = 空/跳過, 其餘為有效流程編號
	ClampA_Setting	: ST_ClampSetting_FeedInToWareHouse;	// A 爪設定 (圓帶來源 + 目的地)
	ClampB_Setting	: ST_ClampSetting_FeedInToWareHouse;	// B 爪設定
END_STRUCT
END_TYPE

// ---- Library/10_Machine/18_HMI_Handshake/OLD_DUTs/ST_FeedInToWareHouseBox_Info.TcDUT
TYPE
    ST_FeedInToWareHouseBox_Info :
    STRUCT
        ClampA_Setting : ST_ClampSetting_FeedInToWareHouse; // Set clampA action (pick from RoundBelt, place to WareHouse)
        ClampB_Setting : ST_ClampSetting_FeedInToWareHouse; // Set clampB action (pick from RoundBelt, place to WareHouse)
    END_STRUCT
END_TYPE

// ---- Library/10_Machine/18_HMI_Handshake/OLD_DUTs/ST_FeedInToWareHouse_Ctrl.TcDUT
TYPE ST_FeedInToWareHouse_Ctrl EXTENDS ST_CommandBasic :
STRUCT
END_STRUCT
END_TYPE

// ---- Library/10_Machine/18_HMI_Handshake/OLD_DUTs/ST_FeedInToWareHouse_Status.TcDUT
TYPE ST_FeedInToWareHouse_Status EXTENDS ST_StatusBasic :
STRUCT
END_STRUCT
END_TYPE

// ---- Library/10_Machine/18_HMI_Handshake/OLD_DUTs/st_FlowBaseCore.TcDUT
TYPE st_FlowBaseCore :
STRUCT
  Start:BOOL;
  Excute:BOOL;
  Done:BOOL;
END_STRUCT
END_TYPE

// ---- Library/10_Machine/18_HMI_Handshake/OLD_DUTs/st_HandshakeBase.TcDUT
TYPE
    st_HandshakeBase :
    STRUCT
        Execute  : BOOL; //觸發命令，持續On到Done出現
        Done     : BOOL; //完成訊號
        Busy     : BOOL; //執行動作中
        Occupied : BOOL; //其他命令執行中，潛在干涉衝突
        Reset    : BOOL; //清除此命令內容
        Error    : BOOL; //錯誤回報
    END_STRUCT
END_TYPE

// ---- Library/10_Machine/18_HMI_Handshake/OLD_DUTs/st_HandShakeBaseWithError.TcDUT
TYPE st_HandShakeBaseWithError:
STRUCT
	stHandShakeBase		:	st_HandshakeBase;
	bError				:	BOOL;
END_STRUCT
END_TYPE

// ---- Library/10_Machine/18_HMI_Handshake/OLD_DUTs/st_ListRunCore.TcDUT
TYPE st_ListRunCore :
STRUCT
	ListRunCore : ARRAY[0..12] OF st_FlowBaseCore;
END_STRUCT
END_TYPE

// ---- Library/10_Machine/18_HMI_Handshake/OLD_DUTs/ST_ManualServoPara.TcDUT
TYPE ST_ManualServoPara :
    STRUCT
        Position :LREAL;
        Velocity :LREAL;
        Distance :LREAL;
        ACC      :LREAL;
        DEC      :LREAL;
        Jerk     :LREAL;
    END_STRUCT
END_TYPE

// ---- Library/10_Machine/18_HMI_Handshake/OLD_DUTs/ST_MechanicalList.TcDUT
TYPE
    ST_MechanicalList :
    STRUCT
        BoxRow : INT := 5; // Number of rows of the box containing drill pins.
        BoxColumn : INT := 10; // Number of columns of the box containing drill pins.
        TableWaitBoxPos : LREAL := 352.2; // Storage SimpleAllocate Table position for load / unload box.
        O5_OffsetData : stPositionCommand; // The position offset of O5 position
		O6_OffsetData : stPositionCommand; // The position offset of O6 position
		O7_OffsetData : stPositionCommand; // The position offset of O7 position
		O8_OffsetData : stPositionCommand; // The position offset of O8 position
    END_STRUCT
END_TYPE

// ---- Library/10_Machine/18_HMI_Handshake/OLD_DUTs/st_ModbusSwitchOff.TcDUT
TYPE st_ModbusSwitchOff :
STRUCT
	switchOff_1 : BOOL :=FALSE;
	switchOff_2 : BOOL :=FALSE;
	switchOff_3 : BOOL :=FALSE;
	switchOff_4 : BOOL :=FALSE;
END_STRUCT
END_TYPE

// ---- Library/10_Machine/18_HMI_Handshake/OLD_DUTs/ST_Mode.TcDUT
TYPE ST_Mode :
STRUCT
	// Mode :  0 : Trainsitioning
	// 		   1 : Manual
	// 		   2 : Auto
	// 		   3 : Service(No implement yet)
	//        99 : ModeSelect
	TargetMode	:E_MachineMode := E_MachineMode.UNDEFINE; 	
	CurrentMode :E_MachineMode:=E_MachineMode.ModeSelect;
	HandshakeBase : st_HandshakeBase;
END_STRUCT
END_TYPE

// ---- Library/10_Machine/18_HMI_Handshake/OLD_DUTs/st_MoveConveyorJob.TcDUT
TYPE st_MoveConveyorJob :
STRUCT
	tTime			: LREAL;	//Time in s
	bMoveReverse	: BOOL;		//Move backward if true
	HandShake		: st_HandshakeBase;
END_STRUCT
END_TYPE

// ---- Library/10_Machine/18_HMI_Handshake/OLD_DUTs/ST_OffsetData.TcDUT
TYPE
    ST_OffsetData :
    STRUCT
        WarehouseA        : ARRAY[1..10, 1..20, 1..2] OF ST_PositionOffsetData; // [x,y,z] X: Layer, Y: Slide, Z: Clamp
        WarehouseB        : ARRAY[1..10, 1..20, 1..2] OF ST_PositionOffsetData; // [x,y,z] X: Layer, Y: Slide, Z: Clamp
        RoundBelt         : ARRAY[1..2, 1..2] OF ST_PositionOffsetData; // [x,y] X: Address, Y: Clamp
        BufferArea        : ARRAY[1..28, 1..2] OF ST_PositionOffsetData; // [x,y] X: Address, Y: Clamp
        LoadConveyor      : ARRAY[1..2, 1..2] OF ST_PositionOffsetData; // [x,y] X: Address, Y: Clamp
        SimpleAllocate    : ARRAY[1..2, 1..2] OF ST_PositionOffsetData; // [x,y] X: Address, Y: Clamp
        InOutConveyor     : ARRAY[1..3, 1..2] OF ST_PositionOffsetData; // [x,y] X: Address, Y: Clamp
        WareHouseA_Buffer : ARRAY[1..2] OF ST_PositionOffsetData; // [x] X: Clamp
        PullOutConveyor   : ARRAY[1..2, 1..2] OF ST_PositionOffsetData; // [x,y] X: Address, Y: Clamp
        ImageInspection   : ARRAY[1..2, 1..2] OF ST_PositionOffsetData; // [x,y] X: Address, Y: Clamp
        DiameterDetect    : ARRAY[1..2, 1..2] OF ST_PositionOffsetData; // [x,y] X: Address, Y: Clamp
    END_STRUCT
END_TYPE

// ---- Library/10_Machine/18_HMI_Handshake/OLD_DUTs/st_OneDirectionCore.TcDUT
TYPE st_OneDirectionCore :
STRUCT
  fname:STRING;
  index:LREAL;
  TargetDistance:LREAL;
  Execute:BOOL;
  Done:BOOL;
END_STRUCT
END_TYPE

// ---- Library/10_Machine/18_HMI_Handshake/OLD_DUTs/ST_OneProcessServoPara.TcDUT
TYPE ST_OneProcessServoPara :
    STRUCT
        Position :LREAL;
        Velocity :LREAL;
        Distance :LREAL;
        ACC      :LREAL;
        DEC      :LREAL;
        Jerk     :LREAL;
    END_STRUCT
END_TYPE

// ---- Library/10_Machine/18_HMI_Handshake/OLD_DUTs/ST_OpPannelStatus.TcDUT
TYPE ST_OpPannelStatus :
    STRUCT
        StartBtnStatus :BOOL; // True : Start botton have been active
        StopBtnStatus  :BOOL; // True : Stop botton have been active
        ResetBtnStatus :BOOL; // True : Reset botton have been active
        EStopBtnStatus :BOOL; // True : EStop botton have been active
		HomeRequestStatus : BOOL; // Home request from panel operator
    END_STRUCT
END_TYPE

// ---- Library/10_Machine/18_HMI_Handshake/OLD_DUTs/st_OutRobotParameterCore.TcDUT
////出料區座標結構
TYPE st_OutRobotParameterCore  :
STRUCT
   fName  :STRING;
   index:  LREAL;
	X      :LREAL;
	Y      :LREAL;
	Rotate :LREAL;
	Clip   :LREAL;
	Excute:BOOL;
	Done  :BOOL;
END_STRUCT
END_TYPE

// ---- Library/10_Machine/18_HMI_Handshake/OLD_DUTs/ST_PositionOffsetData.TcDUT
TYPE ST_PositionOffsetData :
	STRUCT
		Offset_X : REAL; // Fanuc robot X offset distance.
		Offset_Y : REAL; // Fanuc robot Y offset distance.
		Offset_Z : REAL; // Fanuc robot Z offset distance.
		Offset_W : REAL; // Fanuc robot W offset distance.
		Offset_P : REAL; // Fanuc robot P offset distance.
		Offset_R : REAL; // Fanuc robot R offset distance.
	END_STRUCT
END_TYPE

// ---- Library/10_Machine/18_HMI_Handshake/OLD_DUTs/ST_PullOutConveyorInfo.TcDUT
TYPE ST_PullOutConveyorInfo :
STRUCT
	ConveyorRunningTime : TIME; // This variable is the operating time of the conveyor belt forward.
	ConveyorReverseTime : TIME; // This variable is the operating time of the conveyor belt reverse.
	CommandType : E_PullOutConveyorCommandType; // Select PullOut conveyor command.
END_STRUCT
END_TYPE

// ---- Library/10_Machine/18_HMI_Handshake/OLD_DUTs/ST_ReadAllOffsetDataCommand.TcDUT
TYPE ST_ReadAllOffsetDataCommand EXTENDS ST_CommandBasic:
STRUCT
END_STRUCT
END_TYPE

// ---- Library/10_Machine/18_HMI_Handshake/OLD_DUTs/ST_ReadAllOffsetDateStatus.TcDUT
TYPE ST_ReadAllOffsetDateStatus EXTENDS ST_StatusBasic :
STRUCT
END_STRUCT
END_TYPE

// ---- Library/10_Machine/18_HMI_Handshake/OLD_DUTs/ST_ReadSingleOffsetData_Command.TcDUT
TYPE ST_ReadSingleOffsetData_Command EXTENDS ST_CommandBasic :
STRUCT
END_STRUCT
END_TYPE

// ---- Library/10_Machine/18_HMI_Handshake/OLD_DUTs/ST_ReadSingleOffsetData_Info.TcDUT
TYPE ST_ReadSingleOffsetData_Info :
STRUCT
	WareHouse 	: E_WareHouse; 		// Select the target of warehouse. 
	Layer 		: E_WareHouseLayer; // Select the target of layer.
	Slide 		: E_WareHouseSlide; // Select the target of slide.
	Area		: E_RobotArea; // Select the target of area (Abs move)
	Address		: INT; // Select the target of Address (Abs move)
	Clamp		: E_RobotClamp; // 1 :ClampA, 2: ClampB
END_STRUCT
END_TYPE

// ---- Library/10_Machine/18_HMI_Handshake/OLD_DUTs/ST_ReadSingleOffsetData_Status.TcDUT
TYPE ST_ReadSingleOffsetData_Status EXTENDS ST_StatusBasic :
STRUCT
END_STRUCT
END_TYPE

// ---- Library/10_Machine/18_HMI_Handshake/OLD_DUTs/ST_ReloadRoundBeltBox_Info.TcDUT
TYPE
    ST_ReloadRoundBeltBox_Info :
    STRUCT
        ClampA_Setting : ST_ClampSetting_ReloadRoundBelt; // Set clampA action.
        ClampB_Setting : ST_ClampSetting_ReloadRoundBelt; // Set clampB action.
    END_STRUCT
END_TYPE

// ---- Library/10_Machine/18_HMI_Handshake/OLD_DUTs/ST_ReloadRoundBelt_Ctrl.TcDUT
TYPE ST_ReloadRoundBelt_Ctrl EXTENDS ST_CommandBasic :
STRUCT
END_STRUCT
END_TYPE

// ---- Library/10_Machine/18_HMI_Handshake/OLD_DUTs/ST_ReloadRoundBelt_Status.TcDUT
TYPE ST_ReloadRoundBelt_Status EXTENDS ST_StatusBasic :
STRUCT
END_STRUCT
END_TYPE

// ---- Library/10_Machine/18_HMI_Handshake/OLD_DUTs/st_Robot.TcDUT
TYPE st_Robot :
STRUCT
	//Position = XXX~XXX為倉別移動, XXX~XXX為絕對移動
	Position	: UINT;
	//Grabber = 1為夾爪A, Grabber = 2為夾爪B
	Grabber		: UINT;
	//Activity = 1為夾取, Activity = 0為開爪
	Activity	: UINT;
END_STRUCT
END_TYPE

// ---- Library/10_Machine/18_HMI_Handshake/OLD_DUTs/st_RobotMoveAbs.TcDUT
TYPE st_RobotMoveAbs :
STRUCT
	
AbsPositionX : LREAL;
AbsPositionY : LREAL;
AbsPositionR : LREAL; // for allocate robot , R targer position whith no effevt
Execute		 : BOOL;
Done		 : BOOL;
END_STRUCT
END_TYPE

// ---- Library/10_Machine/18_HMI_Handshake/OLD_DUTs/ST_RobotRegionMove_Info.TcDUT
TYPE ST_RobotRegionMove_Info :
STRUCT
	Get				: BOOL;
	UseA			: BOOL;
	UseB			: BOOL;
	A_Position		: LREAL;
	B_Position		: LREAL;
END_STRUCT
END_TYPE

// ---- Library/10_Machine/18_HMI_Handshake/OLD_DUTs/ST_RoundBeltCoordinates.TcDUT
TYPE ST_RoundBeltCoordinates :
STRUCT
	Station : E_RoundBeltStation;
	ReloadCarrier : E_ReloadRoundBelt_PlaceAddress;
END_STRUCT
END_TYPE

// ---- Library/10_Machine/18_HMI_Handshake/OLD_DUTs/st_SafetyByPass.TcDUT
TYPE st_SafetyByPass :
STRUCT
	SafeDoorByPass :BOOL := FALSE;
	//AliveCheckingBYPass : BOOL;
END_STRUCT
END_TYPE

// ---- Library/10_Machine/18_HMI_Handshake/OLD_DUTs/ST_SaveParaDefault.TcDUT
TYPE
    ST_SaveParaDefault :
    STRUCT
        Command : ST_CommandBasic;
        Status  : ST_StatusBasic;
    END_STRUCT
END_TYPE

// ---- Library/10_Machine/18_HMI_Handshake/OLD_DUTs/ST_SaveParaRemote.TcDUT
TYPE
    ST_SaveParaRemote :
    STRUCT
        Command : ST_CommandBasic;
        Status  : ST_StatusBasic;
    END_STRUCT
END_TYPE

// ---- Library/10_Machine/18_HMI_Handshake/OLD_DUTs/st_ServiceTimeoutSetting.TcDUT
TYPE st_ServiceTimeoutSetting :
STRUCT
	tRobotMovementTimeout	 : INT := 60000; // Time in ms
	tOutRobotPendingForConveyorTimeout : INT := 50000;
END_STRUCT
END_TYPE

// ---- Library/10_Machine/18_HMI_Handshake/OLD_DUTs/ST_ServoList.TcDUT
TYPE ST_ServoList :
STRUCT
	TableAxis : ST_ServoParaBasic;
END_STRUCT
END_TYPE

// ---- Library/10_Machine/18_HMI_Handshake/OLD_DUTs/ST_ServoParaBasic.TcDUT
TYPE ST_ServoParaBasic :
    STRUCT
        ManualMode     :ST_ManualServoPara;
        AutoMode       :ST_AutoServoPara;
        OneProcessMode :ST_OneProcessServoPara;
    END_STRUCT
END_TYPE

// ---- Library/10_Machine/18_HMI_Handshake/OLD_DUTs/ST_SimpleAllocateCommand.TcDUT
TYPE ST_SimpleAllocateCommand EXTENDS ST_CommandBasic:
    STRUCT
    END_STRUCT
END_TYPE

// ---- Library/10_Machine/18_HMI_Handshake/OLD_DUTs/ST_SimpleAllocateInfo.TcDUT
TYPE ST_SimpleAllocateInfo :
    STRUCT
        PickBox     :E_SimpleAllocateTable; // Specify the index of the box to pick up.
        PlaceBox    :E_SimpleAllocateTable; // Specify the index of the box to place.
        PickIndex_X :E_HoleIndex_X; // Specify the starting column index to pick up the drill pin.
        PickIndex_Y :E_HoleIndex_Y; // Specify the starting row index to pick up the drill pin.
        PickAmount  :INT;
		TableHolePos	: ARRAY[1..4] OF LREAL; // Simple Allocate Axis has 4 hole, set the 4 hole position
    END_STRUCT
END_TYPE

// ---- Library/10_Machine/18_HMI_Handshake/OLD_DUTs/ST_SimpleAllocateStatus.TcDUT
TYPE ST_SimpleAllocateStatus EXTENDS ST_StatusBasic:
    STRUCT
    END_STRUCT
END_TYPE

// ---- Library/10_Machine/18_HMI_Handshake/OLD_DUTs/st_SixAxisRobotCore.TcDUT
TYPE st_SixAxisRobotCore :
STRUCT
	WDataCore:st_AutoSixAxisWarehouseParameter;
	AbslutCore:st_AutoSixAxisAbsMoveParameter;
END_STRUCT
END_TYPE

// ---- Library/10_Machine/18_HMI_Handshake/OLD_DUTs/st_SixAxisWarehouseParameter.TcDUT
TYPE st_SixAxisWarehouseParameter  :
STRUCT
	Warehouse:LREAL; //WarehouseA = 1, WarehouseB = 0
	Layer : LREAL;
	Slide : LREAL;	
	Clip:LREAL;
	Get:BOOL;	//出盒
	Push:BOOL;	//入盒
	Excute:BOOL;
	Done  :BOOL;
	Busy  : BOOL;
	Occupied : BOOL;
//	Error : BOOL;
END_STRUCT
END_TYPE

// ---- Library/10_Machine/18_HMI_Handshake/OLD_DUTs/st_StationPositions.TcDUT
TYPE st_StationPositions :
STRUCT
	Position : LREAL;
END_STRUCT
END_TYPE

// ---- Library/10_Machine/18_HMI_Handshake/OLD_DUTs/ST_StatusBasic.TcDUT
TYPE ST_StatusBasic :
STRUCT
    Busy	:BOOL;	// TRUE : Process is running
    Done	:BOOL;	// TRUE : Process is done
    Error	:BOOL;	// TRUE : Process has error
	//ErrorID :UINT;
	Status : T_MaxString; // Show the error msg
END_STRUCT
END_TYPE

// ---- Library/10_Machine/18_HMI_Handshake/OLD_DUTs/ST_SystemParameter.TcDUT
TYPE ST_SystemParameter :
STRUCT
	Cylinder : ST_CylinderList;
	Servo : ST_ServoList;
	Mechanical : ST_MechanicalList;
	//Motor :ST_MotorList;
END_STRUCT
END_TYPE

// ---- Library/10_Machine/18_HMI_Handshake/OLD_DUTs/ST_WareHouseCoordinates.TcDUT
TYPE ST_WareHouseCoordinates :
STRUCT
	Layer : E_WareHouseLayer;
	Slide : E_WareHouseSlide;
END_STRUCT
END_TYPE

// ---- Library/10_Machine/18_HMI_Handshake/OLD_DUTs/ST_WareHouseInnerPickBatch.TcDUT
// 倉儲內取放圓帶 — 批次結構
// 最多 40 筆流程，由上位機 (C# HMI) 透過 ADS 寫入 FlowInfo 陣列
// HandShake 控制啟動 (Execute) / 完成 (Done) / 錯誤 (Error) / 重置 (Reset)
// WorkedID 回報每筆流程完成狀態 → C# 端據此更新 SQL 紀錄
// ActionRecords 為每筆流程的倉儲取放紀錄，C# 透過 FeedBack 握手讀取
TYPE ST_WareHouseInnerPickBatch :
STRUCT
	FlowInfo		: ARRAY[0..39] OF ST_WareHouseInnerPickFlowInfo;	// 流程陣列，最多 40 筆
	HandShake		: st_HandshakeBase;		// Execute/Done/Busy/Error/Reset 握手信號
	NrOfFlow		: UINT;		// 本次批次有效流程數量 (0..40)
	Pause			: BOOL;		// TRUE = 暫停批次執行 (完成當前流程後暫停)
	WorkedID		: ARRAY[0..39] OF INT;	// 完成回報：-1 = 未完成, 其餘 = 已完成的流程 ID
	ActionRecords	: ARRAY[0..39] OF ST_ClampActionRecord;	// 當前流程的倉儲取放動作紀錄
	ActionIndex		: INT;		// 已記錄筆數
	FeedBack		: BOOL;		// PLC → C#: 陣列可讀取
	ReadComplete	: BOOL;		// C# → PLC: 讀取完成確認
END_STRUCT
END_TYPE

// ---- Library/10_Machine/18_HMI_Handshake/OLD_DUTs/ST_WareHouseInnerPickFlowInfo.TcDUT
// 倉儲內取放圓帶 — 單筆流程資訊
// 定義 A/B 爪各自的倉儲來源、圓帶目標、以及要取的目標深度 (Position)
// 由上位機 (C# HMI) 透過 ADS 寫入，PLC 端根據此結構執行取放動作
//
// TargetPosition 說明：
//   1 = P1 = 最前面的盒子 (直接取)
//   2 = P2 = 第二個盒子 (需協助爪搬開 P1)
//   3+ = P3 以後 (需先清除前面盒子到 buffer，再由協助爪配合目標爪取放)
//   0 = 不使用此爪
TYPE ST_WareHouseInnerPickFlowInfo :
STRUCT
	ID				: INT := -1;	// 流程 ID, -1 = 空/跳過, 其餘為有效流程編號
	ClampA_Setting	: ST_ClampSetting_ReloadRoundBelt;	// A 爪設定：倉儲來源 (倉別/層/軌) + 圓帶目標 (站位/載具)
	ClampB_Setting	: ST_ClampSetting_ReloadRoundBelt;	// B 爪設定：倉儲來源 (倉別/層/軌) + 圓帶目標 (站位/載具)
	TargetPositionA	: INT;	// A 爪目標深度 1..10, 0 = 此爪不動作
	TargetPositionB	: INT;	// B 爪目標深度 1..10, 0 = 此爪不動作
END_STRUCT
END_TYPE

// ---- Library/10_Machine/18_HMI_Handshake/OLD_DUTs/ST_WriteAllOffsetData_Command.TcDUT
TYPE ST_WriteAllOffsetData_Command EXTENDS ST_CommandBasic :
STRUCT
END_STRUCT
END_TYPE

// ---- Library/10_Machine/18_HMI_Handshake/OLD_DUTs/ST_WriteAllOffsetData_Info.TcDUT
TYPE ST_WriteAllOffsetData_Info EXTENDS ST_StatusBasic :
STRUCT
END_STRUCT
END_TYPE

// ---- Library/10_Machine/18_HMI_Handshake/OLD_DUTs/ST_WriteAllOffsetData_Status.TcDUT
TYPE ST_WriteAllOffsetData_Status EXTENDS ST_StatusBasic :
STRUCT
END_STRUCT
END_TYPE

// ---- Library/10_Machine/18_HMI_Handshake/OLD_DUTs/ST_WriteSingleOffsetData_Command.TcDUT
TYPE ST_WriteSingleOffsetData_Command EXTENDS ST_CommandBasic :
STRUCT
END_STRUCT
END_TYPE

// ---- Library/10_Machine/18_HMI_Handshake/OLD_DUTs/ST_WriteSingleOffsetData_Info.TcDUT
TYPE ST_WriteSingleOffsetData_Info :
STRUCT
	WareHouse 	: E_WareHouse; 		// Select the target of warehouse. 
	Layer 		: E_WareHouseLayer; // Select the target of layer.
	Slide 		: E_WareHouseSlide; // Select the target of slide.
	Area		: E_RobotArea; // Select the target of area (Abs move)
	Address		: INT; // Select the target of Address (Abs move)
	Clamp		: E_RobotClamp; // 1 :ClampA, 2: ClampB
END_STRUCT
END_TYPE

// ---- Library/10_Machine/18_HMI_Handshake/OLD_DUTs/ST_WriteSingleOffsetData_Status.TcDUT
TYPE ST_WriteSingleOffsetData_Status EXTENDS ST_StatusBasic :
STRUCT
END_STRUCT
END_TYPE

// ---- Library/10_Machine/18_HMI_Handshake/Service/DUTs/ST_HMI_Handshake.TcDUT
TYPE
    ST_HMI_Handshake :
    STRUCT
      //========單動一行程============
	// one process use
    //配針單動資料結構
    AllocateMoveStructure : REFERENCE TO st_ads_AllocateMoveStructure;
	//拔針單動資料結構
    AllocateMoveStructure_Reverse : REFERENCE TO st_ads_AllocateMoveStructure;     
    //空盒手臂單動資料結構
    EmptyRobotToTurnTableMove : REFERENCE TO st_ads_OneAxisMoveWithPosition;
    //圓帶單動一行程
    AllocateCircleMove : REFERENCE TO st_AllocateCircleMoveStructure;
    //圓盤單動一行程
    TurnTableMove : REFERENCE TO st_ads_OneAxisMoveWithPosition;
//    //軸還原預設狀態
//    AxesControl : REFERENCE TO ARRAY[0..10] OF st_AxisControl;
    //機台還原預設狀態
    MachineReset : REFERENCE TO st_ads_MachineReset;
    //Empty
    RareFullBoxPush : REFERENCE TO st_ads_OutRobtToPlateMove;
		// Move Allocate robot to needling position
	AllocationRobotNeedlingMove : REFERENCE TO st_AllocateRobotNeedlingMove;

//==============自動模式=========================

    //AutoModeUse*-------自動模式圓帶單動
    AutoMode_AllocateCircleMove : REFERENCE TO st_AllocateCircleMoveStructure;
    //AutoModeUse*-------手臂倉儲位置移動
    AutoMode_RobotWarehouseMove : REFERENCE TO st_AutoSixAxisWarehouseParameter;
    //AutoModeUse*-------手臂絕對位置移動
    AutoMode_RobotAbsMove : REFERENCE TO st_AutoSixAxisAbsMoveParameter;
    //AutoModeUse*-------空盒取料移動
    AutoMode_EmptyBoxMove : REFERENCE TO st_AutoMode_ClampingBoxesJob;
    //AutoModeUse*-------圓盤移動
    AutoMode_TurnTableMOve : REFERENCE TO st_ads_OneAxisMoveWithPosition;
    //AutoModeUse--------配針
    AutoMode_AllocateMove : REFERENCE TO st_AutoMode_AllocatingJob;
	 //AutoModeUse--------拔針
    AutoMode_AllocateMove_Reverse : REFERENCE TO st_AutoMode_AllocatingJob;
	//AutoModeUse--------配針batch mode
	AutoMode_AllocateBatchMode	: REFERENCE TO ST_AllocationJobBatchMode;
	//AutoModeUse--------拔針batch mode
	AutoMode_AllocateBatchMode_Reverse	: REFERENCE TO ST_AllocationJobBatchMode;
	//AutoModeSimpleAllocation_Batch
	AutoMode_SimpleAllocation_Batch		: REFERENCE TO ST_AllocationJobBatchMode;
    //AutoMdeUse---------散針放盒
    AutoMode_RareBoxMove : REFERENCE TO st_AutoMode_ClampingBoxesJob;
    //AutoMdeUse---------出貨放盒單動
    AutoMode_OutBoxMove : REFERENCE TO st_AutoMode_ClampingToPlate;
	//AutoMdeUse---------拔針放盒自動模式
    AutoMode_BoxMoveReverse : REFERENCE TO st_AutoMode_ClampingBoxesJob;
    //倉儲分選區移動,移動位置列表需延伸此陣列取得 WarehouseMovePosition :ARRAY[0..3] OF st_OneDirectionCore;
    AutoMode_WarehouseMove : REFERENCE TO st_ads_OneAxisMoveWithPosition;
    //AutoModeUse------手臂區域移動_FeedIn conveyor
	AutoMode_RobotRegionMove_FeedInConveyor		: REFERENCE TO ST_AutoMode_RobotRegionMove;
	//AutoModeUse------手臂區域移動_AllocatedConveyor
	AutoMode_RobotRegionMove_AllocatedConveyor		: REFERENCE TO ST_AutoMode_RobotRegionMove;
	//AutoModeUse------手臂區域移動_Pullout conveyor
	AutoMode_RobotRegionMove_PullOutConveyor		: REFERENCE TO ST_AutoMode_RobotRegionMove;
	//AutoModeUse------手臂區域移動_Buffer area
	AutoMode_RobotRegionMove_BufferArea		: REFERENCE TO ST_AutoMode_RobotRegionMove;
	//AutoModeUse------手臂區域移動_RoundBelt
	AutoMode_RobotRegionMove_RoundBelt		: REFERENCE TO ST_AutoMode_RobotRegionMove;
   //AutoMode MoveConveyorJob------定時移動輸送帶
    AutoMode_MoveConveyorJob : REFERENCE TO st_MoveConveyorJob;
	// Automode Feedin empty box with robot 
	AutoMode_FeedInEmptyBoxWithRobot : REFERENCE TO ST_AutoMode_FeedInEmptyBox; // Automode : Feedin empty box with robot from Warehouse and Pullout convenyor
	// Automode Reload RoundBelt box with robot
	AutoMode_ReloadRoundBeltBoxWithRobot : REFERENCE TO ST_AutoMode_ReloadRoundBeltBox; // Automode : Reload RoundBelt box with robot from warehouse
	// Automode FeedIn RoundBelt box to warehouse - 圓帶到倉儲
	AutoMode_FeedInRoundBeltBoxToWareHouse : REFERENCE TO ST_AutoMode_FeedInToWareHouseBox; // Automode : Pick box from RoundBelt and place to WareHouse
	//AutoMode UpperFeedInConveyor
	AutoMode_UpperFeedInConveyor : REFERENCE TO ST_Auto_UpperFeedInConveyor;
	//AutoModeUse------倉儲馬達搭配手臂移動
    AutoMode_WarehouseMotoWithRobotMove : REFERENCE TO st_AutoSixAxisWarehouseParameter;
    //SimpleAllocate Autode-----簡易配針
	AutoMode_SimpleAllocate    : REFERENCE TO ST_AutoMode_SimpleAllocateHandShake; // AutoMode Simple Allocate
    AutoMode_PullOutConveyor   : REFERENCE TO ST_AutoPullOutConveyor; // AutoMode PullOut Conveyor
    //AutoModeUse----------錯誤通知  Host To PLC
    AutoMode_ErrorHandle : REFERENCE TO st_Alarm;
    //Alarm report	----------錯誤通知 PLC to Host
    AlarmAllocation : REFERENCE TO ARRAY[0..999] OF ST_Alarm_Tmax;
	//AutoMode Use------ShippingGoodV2		20250304 Min
	AutoMode_AddBoxes	: REFERENCE TO ST_AutoAddsBoxes;
    //=================TwinCat Memory============
    //TwinCatMemory				:st_TwinCatMemory;
    //=================全局Home===================

    MachineHome          : REFERENCE TO st_RegionHome; // Machine all units home command
    StorageRegionHome    : REFERENCE TO st_RegionHome;
    AllocationRegionHome : REFERENCE TO st_RegionHome;
    FGARegionHome        : REFERENCE TO st_RegionHome;

    //===============手自動=======================
    StorageRegionMode : REFERENCE TO ST_Mode;
    AllocationRegion  : REFERENCE TO ST_Mode;
    FGARegionMode     : REFERENCE TO ST_Mode;
    MachineMode       : REFERENCE TO ST_Mode;
	
    // Operation Pannel Status
    OpPannel_Status : REFERENCE TO ST_OpPannelStatus; //PLC -> HMI
    OpPannel_Ctrl   : REFERENCE TO ST_OpPannelStatus; // HMI -> PLC

	//20250425 addon
	//Machine state
//	MachineState : REFERENCE TO E_MachineState;
	
	FanucRobot_General               : REFERENCE TO ST_FanucRobotGeneralCtrl;
	
	//AutoModeUse------倉儲小手臂ABS 移動
	AutoMode_ShippingRobot_Left            : REFERENCE TO ST_AutoMode_ShippingRobot_MoveAbs;
	//AutoModeUse------倉儲小手臂ABS 移動
	AutoMode_ShippingRobot_Right           :REFERENCE TO  ST_AutoMode_ShippingRobot_MoveAbs;
	//AutoModeUse------倉儲小手臂ABS 移動
	AutoMode_ShippingRobot_TransmitCVEnd    : REFERENCE TO ST_AutoMode_ShippingRobot_MoveAbs;
	//AutoModeUse------同尺寸拍照
	AutoMode_SameSizeCVCamera				: REFERENCE TO ST_AutoMode_TransCVCamera;
	//AutoModeUse------同尺寸反向拍照
	AutoMode_SameSizeCVCamera_Reverse		: REFERENCE TO ST_AutoMode_TransCVCamera;
	//AutoModeUse------不同尺寸拍照
	AutoMode_DifferentCVCamera				: REFERENCE TO ST_AutoMode_TransCVCamera;
	
	//AutoModeUse------倉儲內取放圓帶 (單筆)
	AutoMode_WareHouseInnerPickToRoundBelt		: REFERENCE TO ST_AutoMode_WareHouseInnerPickToRoundBelt;
	//AutoModeUse------倉儲內取放圓帶 (批次)
	AutoMode_WareHouseInnerPickToRoundBeltBatch	: REFERENCE TO ST_WareHouseInnerPickBatch;
	//AutoModeUse------圓帶回倉/PullOut (批次)
	AutoMode_FeedInRoundBeltBoxBatch			: REFERENCE TO ST_FeedInRBBatch;
	//Reboot Modbus devices
	RebootModbusDevices			: REFERENCE TO st_RebootModbusDevices;
	
	//Shipping FeedOut TransCV with HansLaser handshake Service
	AutoMode_ShippingLeftSideTransCV			: REFERENCE TO ST_AutoMode_ShippingLeftSideTransCV;
	AutoMode_ShippingRightSideTransCV			: REFERENCE TO ST_AutoMode_ShippingRightSideTransCV;

	//AutoModeUse------- 出貨區緩衝區
	AutoMode_ShippingRobot_Buffer			:REFERENCE TO ST_AutoMode_ShippingRobot_MoveAbs;
	//AutoModeUse------- 出貨區拍照位置		
	AutoMode_ShippingRobot_PhotoStandByPos	:REFERENCE TO ST_AutoMode_ShippingRobot_MoveAbs;
	//AutoModeUse------- 出貨區搬運 (合併)
	AutoMode_ShippingRobotTransfer			:REFERENCE TO ST_AutoMode_ShippingRobotTransfer;
	//AutoModeUse------- 出貨區小手臂鐵盤掃描
	AutoMode_ShippingPlateScan				: REFERENCE TO ST_ShippingPlateToConveyor;
	//AutoMode---------- 倉儲區手臂單獨回原點
	AutoMode_RobotSelfHoming				: REFERENCE to ST_AutoMode_RobotSelfHoming;
	//AutoModeUse------逆向拍照批次入料
	AutoMode_ReverseBatchPick				: REFERENCE TO ST_AutoMode_ReverseBatchPick;
	//AutoModeUse------同尺寸軌道回倉/NG
	AutoMode_ReverseBoxToWareHouse			: REFERENCE TO ST_AutoMode_ReverseBoxToWareHouse;
	//BuzzCtrl
	BuzzCtrl								: REFERENCE TO ST_BuzzCtrl;
			
    END_STRUCT
END_TYPE

// ---- Library/10_Machine/19_Device/EL1889/ST_InputTable.TcDUT
TYPE
    ST_InputTable :
    STRUCT
        bUpCV_BoxArrived_Sensor                       : BIT; //X6.0
        bUpCV_Block1Detect_Sensor                     : BIT; //X6.1
        bUpCV_Block2Detect_Sensor                     : BIT; //X6.2
        bUpCV_Block3Detect_Sensor                     : BIT; //X6.3
        bUpCV_ReLoadDetect_Sensor                     : BIT; //X6.4
        bUpCV_Block1_RearSensor                       : BIT; //X6.5
        bUpCV_Block2_RearSensor                       : BIT; //X6.6
        bUpCV_Block3_RearSensor                       : BIT; //X6.7
        bLowCV_BoxArrived_Sensor                      : BIT; //X6.8
        bLowCV_Block1Detect_Sensor                    : BIT; //X6.9
        bLowCV_Block2Detect_Sensor                    : BIT; //X6.10
        bLowCV_Block1_RearSensor                      : BIT; //X6.11
        bLowCV_Block2_RearSensor                      : BIT; //X6.12
        bLowCV_2ndBoxGap_Sensor                       : BIT; //X6.13
        spare15                                       : BIT; //X6.14
        spare16                                       : BIT; //X6.15
        bUpCV_DiameterHoriz_FrontSensor               : BIT; //X7.0
        bUpCV_DiameterHoriz_RearSensor                : BIT; //X7.1
        bUpCV_DiameterVert_FrontSensor                : BIT; //X7.2
        bUpCV_DiameterVert_RearSensor                 : BIT; //X7.3
        spare21                                       : BIT; //X7.4
        spare22                                       : BIT; //X7.5
        spare23                                       : BIT; //X7.6
        spare24                                       : BIT; //X7.7
        spare25                                       : BIT; //X7.8
        spare26                                       : BIT; //X7.9
        bStorage_AirPressure_Ready                    : BIT; //X7.10
        bStorage_EstopPb                              : BIT; //X7.11
        bStorage_StartPb                              : BIT; //X7.12
        bStorage_StopPb                               : BIT; //X7.13
        bStorage_ResetPb                              : BIT; //X7.14
        spare32				                          : BIT; //X7.15
        bStackPush_DCMotor_PosLimit                   : BIT; //X9.0
        bStackPush_DCMotor_NegLimit                   : BIT; //X9.1
        bStackPush_Pusher_FrontSensor                 : BIT; //X9.2
        bStackPush_Pusher_RearSensor                  : BIT; //X9.3
        bStorage_StackPushPb                          : BIT; //X9.4
        Spare38                                       : BIT; //X9.5
        Spare39                                       : BIT; //X9.6
        Spare40                                       : BIT; //X9.7
        bPullOutCV_AsideEntry_Sensor                  : BIT; //X9.8
        bPullOutCV_AsideExit_Sensor                   : BIT; //X9.9
        bPullOutCV_Aside2ndBoxGap_Sensor              : BIT; //X9.10
        bPullOutCV_BsideEntry_Sensor                  : BIT; //X9.11
        bPullOutCV_BsideExit_Sensor                   : BIT; //X9.12
        bPullOutCV_Bside2ndBoxGap_Sensor              : BIT; //X9.13
        bPullOutCV_AsideBlock_RearSensor              : BIT; //X9.14
        bPullOutCV_BsideBlock_RearSensor              : BIT; //X9.15
        bSafetyDoor1                                  : BIT; //X10.0
        bSafetyDoor2                                  : BIT; //X10.1
        bSafetyDoor14                                 : BIT; //X10.2
        Spare52                                       : BIT; //X10.3
        bSafetyDoor13                                 : BIT; //X10.4
        bSafetyDoor12                                 : BIT; //X10.5
        bSafetyDoor11                                 : BIT; //X10.6
        bSafetyDoor10                                 : BIT; //X10.7
        bSafetyDoor9                                  : BIT; //X10.8
        spare58                                       : BIT; //X10.9
        spare59                                       : BIT; //X10.10
        spare60                                       : BIT; //X10.11
        spare61                                       : BIT; //X10.12
        spare62                                       : BIT; //X10.13
        bPullOutCV_FwdPb                              : BIT; //X10.14
        bPullOutCV_RevPb                              : BIT; //X10.15
        bAllocateRobot_LeftVert1_HighSensor           : BIT; //X0.0
        bAllocateRobot_LeftVert1_LowSensor            : BIT; //X0.1
        bAllocateRobot_LeftVert2_HighSensor           : BIT; //X0.2
        bAllocateRobot_LeftVert2_LowSensor            : BIT; //X0.3
        bAllocateRobot_RightVert1_HighSensor          : BIT; //X0.4
        bAllocateRobot_RightVert1_LowSensor           : BIT; //X0.5
        bAllocateRobot_RightVert2_HighSensor          : BIT; //X0.6
        bAllocateRobot_RightVert2_LowSensor           : BIT; //X0.7
        bRoundBelt_ChangeZoneA2Detect_Sensor          : BIT; //X0.8
        bRoundBelt_ChangeZoneA3Detect_Sensor          : BIT; //X0.9
        bRoundBelt_ChangeZonePlug_FrontSensor         : BIT; //X0.10
        bRoundBelt_ChangeZonePlug_RearSensor          : BIT; //X0.11
        bRoundBelt_WorkZoneQ1Detect_Sensor            : BIT; //X0.12
        bRoundBelt_WorkZoneQ2Detect_Sensor            : BIT; //X0.13
        bRoundBelt_WorkZonePlug_FrontSensor           : BIT; //X0.14
        bRoundBelt_WorkZonePlug_RearSensor            : BIT; //X0.15
        bRoundBelt_WorkZonePress_RearSensor           : BIT; //X1.0
        bTempZoneA_Sensor                             : BIT; //X1.1
        bTempZoneB_Sensor                             : BIT; //X1.2
        bTempZoneC_Sensor                             : BIT; //X1.3
        bTempZoneD_Sensor                             : BIT; //X1.4
        bTurnTable_Press_RearSensor                   : BIT; //X1.5
        bTurnTable_R1Detect_Sensor                    : BIT; //X1.6
        bTurnTable_R2Detect_Sensor                    : BIT; //X1.7
        bTurnTable_I2Detect_Sensor                    : BIT; //X1.8
        bTurnTable_I1Detect_Sensor                    : BIT; //X1.9
        bOutRobot_Xaxis_PosLimit                      : BIT; //X1.10
        bOutRobot_Xaxis_HomeSensor                    : BIT; //X1.11
        bOutRobot_Xaxis_NegLimit                      : BIT; //X1.12
        bOutRobot_Yaxis_PosLimit                      : BIT; //X1.13
        bOutRobot_Yaxis_HomeSensor                    : BIT; //X1.14
        bOutRobot_Yaxis_NegLimit                      : BIT; //X1.15
        bOutRobot_AsideVert_HighSensor                : BIT; //X2.0
        bOutRobot_AsideVert_LowSensor                 : BIT; //X2.1
        bOutRobot_BsideVert_HighSensor                : BIT; //X2.2
        bOutRobot_BsideVert_LowSensor                 : BIT; //X2.3
        bOutRobot_AsideClamp_RearSensor               : BIT; //X2.4
        bOutRobot_BsideClamp_RearSensor               : BIT; //X2.5
        spare103                                      : BIT; //X2.6
        bSafetyDoor5			                      : BIT; //X2.7
        spare105                                      : BIT; //X2.8
        bSafetyDoor3                                  : BIT; //X2.9
        bAllocate_Electrical_Cabinet_SafetyDoor       : BIT; //X2.10
        bAllocate_AirPressure_Ready                   : BIT; //X2.11
        bAllocate_StartPb                             : BIT; //X2.12
        bAllocate_StopPb                              : BIT; //X2.13
        bAllocate_ResetPb                             : BIT; //X2.14
        bAllocate_EStopPb                             : BIT; //X2.15
        bSameSizeCV_BoxNearStorageSensor              : BIT; //X3.0
        bDifferentSizeCV_BoxDetect7_Sensor            : BIT; //X3.1
        bDifferentSizeCV_BoxDetect6_Sensor            : BIT; //X3.2
        bDifferentSizeCV_BoxDetect5_Sensor            : BIT; //X3.3
        bDifferentSizeCV_BoxDetect4_Sensor            : BIT; //X3.4
        bTransmit_CamaraHorizDifferentSizeSide_Sensor : BIT; //X3.5
        bTransmit_CamaraHorizSameSizeSide_Sensor      : BIT; //X3.6
        bDifferentSizeCV_BoxDetect3_Sensor            : BIT; //X3.7
        bDifferentSizeCV_BoxDetect2_Sensor            : BIT; //X3.8
        bDifferentSizeCV_BoxDetect1_Sensor            : BIT; //X3.9
        bDifferentSizeCV_BoxNearShippingSensor        : BIT; //X3.10
        bSameSizeCV_BoxDetect6_Sensor                 : BIT; //X3.11
        bSameSizeCV_BoxDetect5_Sensor                 : BIT; //X3.12
        bSameSizeCV_BoxDetect4_Sensor                 : BIT; //X3.13
        Spare127                                      : BIT; //X3.14
        bSameSizeCV_BoxDetect3_Sensor                 : BIT; //X3.15
        bRoundBelt_TransmitCVZonePlug_RearSensor      : BIT; //X8.0
        bRoundBelt_TransmitCVZonePlug_FrontSensor     : BIT; //X8.1
        bRoundBelt_Axis_HomeSensor                    : BIT; //X8.2
        spare132	                                  : BIT; //X8.3
        bSafetyDoor7   		                          : BIT; //X8.4
        bSafetyDoor8           		                  : BIT; //X8.5
        bShippingRobot_ElectricalCabinet_SafetyDoor    : BIT; //X8.6
        bSafetyDoor6                       		      : BIT; //X8.7
        spare137	                                  : BIT; //X8.8
        bTurnTable_Axis_HomeSensor                    : BIT; //X8.9
        bAllocateRobot_Xaxis_PosLimit                 : BIT; //X8.10
        bAllocateRobot_Xaxis_NegLimit                 : BIT; //X8.11
        bSafetyDoor4                                  : BIT; //X8.12
        bSameSizeCV_BoxDetect1_Sensor                 : BIT; //X8.13
        bSameSizeCV_BoxNearShippingSensor             : BIT; //X8.14
        bSameSizeCV_BoxDetect2_Sensor                 : BIT; //X8.15
        bDifferentCV_Block_RearSensor                 : BIT; //X11.0
        bSameSizeCVBlock1_RearSensor                  : BIT; //X11.1
        bSameSizeCVBlock2_RearSensor                  : BIT; //X11.2
        spare148                                      : BIT; //X11.3
        spare149                                      : BIT; //X11.4
        spare150                                      : BIT; //X11.5
        spare151                                      : BIT; //X11.6
        spare152                                      : BIT; //X11.7
        spare153                                      : BIT; //X11.8
        spare154                                      : BIT; //X11.9
        spare155                                      : BIT; //X11.10
        spare156                                      : BIT; //X11.11
        spare157                                      : BIT; //X11.12
        spare158                                      : BIT; //X11.13
        spare159                                      : BIT; //X11.14
        spare160                                      : BIT; //X11.15
        spare161                      				  : BIT; //X4.0
        bShippingTransCV_Rightside_Arrived            : BIT; //X4.1		// 大族給我方的左邊到位訊號，
        spare163						              : BIT; //X4.2
        bShippingTransCV_Leftside_Arrived             : BIT; //X4.3		// 大族給我方的左邊到位訊號，
        spare165                                      : BIT; //X4.4
        bHansLaserMachineError                        : BIT; //X4.5		// 大族給我方的機台錯誤訊號
        spare167                                      : BIT; //X4.6
        spare168                                      : BIT; //X4.7
        spare169                                      : BIT; //X4.8
        spare170                                      : BIT; //X4.9
        spare171                                      : BIT; //X4.10
        spare172                                      : BIT; //X4.11
        spare173                                      : BIT; //X4.12
        spare174                                      : BIT; //X4.13
        spare175                                      : BIT; //X4.14
        spare176                                      : BIT; //X4.15
    END_STRUCT
END_TYPE

// ---- Library/10_Machine/19_Device/EL2889/ST_OutputTable.TcDUT
TYPE
    ST_OutputTable :
    STRUCT
        bUpCV_FeedInPress1_Valve                   : BIT; //Y4.0
        bUpCV_FeedInPress2_Valve                   : BIT; //Y4.1
        bUpCV_DiameterPress_Valve                  : BIT; //Y4.2
        bUpCV_CamaraPress1_Valve                   : BIT; //Y4.3
        bUpCV_CamaraPress2_Valve                   : BIT; //Y4.4
        bUpCV_CamaraPress3_Valve                   : BIT; //Y4.5
        bUpCV_CamaraPress4_Valve                   : BIT; //Y4.6
        bUpCV_Block1_Up_Valve                      : BIT; //Y4.7
        bUpCV_Block1_Down_Valve                    : BIT; //Y4.8
        bUpCV_Block2_Up_Valve                      : BIT; //Y4.9
        bUpCV_Block2_Down_Valve                    : BIT; //Y4.10
        bUpCV_Block3_Up_Valve                      : BIT; //Y4.11
        bUpCV_Block3_Down_Valve                    : BIT; //Y4.12
        Spare14                                    : BIT; //Y4.13
        Spare15                                    : BIT; //Y4.14
        Spare16                                    : BIT; //Y4.15
        bWareHouseCV10_Fwd                         : BIT; //Y5.0
        bWareHouseCV10_Rev                         : BIT; //Y5.1
        bWareHouseCV9_Fwd                          : BIT; //Y5.2
        bWareHouseCV9_Rev                          : BIT; //Y5.3
        bWareHouseCV8_Fwd                          : BIT; //Y5.4
        bWareHouseCV8_Rev                          : BIT; //Y5.5
        bWareHouseCV7_Fwd                          : BIT; //Y5.6
        bWareHouseCV7_Rev                          : BIT; //Y5.7
        bWareHouseCV6_Fwd                          : BIT; //Y5.8
        bWareHouseCV6_Rev                          : BIT; //Y5.9
        bWareHouseCV5_Fwd                          : BIT; //Y5.10
        bWareHouseCV5_Rev                          : BIT; //Y5.11
        bWareHouseCV4_Fwd                          : BIT; //Y5.12
        bWareHouseCV4_Rev                          : BIT; //Y5.13
        bWareHouseCV3_Fwd                          : BIT; //Y5.14
        bWareHouseCV3_Rev                          : BIT; //Y5.15
        bWareHouseCV2_Fwd                          : BIT; //Y6.0
        bWareHouseCV2_Rev                          : BIT; //Y6.1
        bWareHouseCV1_Fwd                          : BIT; //Y6.2
        bWareHouseCV1_Rev                          : BIT; //Y6.3
        bWareHouseCV20_Fwd                         : BIT; //Y6.4
        bWareHouseCV20_Rev                         : BIT; //Y6.5
        bWareHouseCV19_Fwd                         : BIT; //Y6.6
        bWareHouseCV19_Rev                         : BIT; //Y6.7
        bWareHouseCV18_Fwd                         : BIT; //Y6.8
        bWareHouseCV18_Rev                         : BIT; //Y6.9
        bWareHouseCV17_Fwd                         : BIT; //Y6.10
        bWareHouseCV17_Rev                         : BIT; //Y6.11
        bWareHouseCV16_Fwd                         : BIT; //Y6.12
        bWareHouseCV16_Rev                         : BIT; //Y6.13
        bWareHouseCV15_Fwd                         : BIT; //Y6.14
        bWareHouseCV15_Rev                         : BIT; //Y6.15
        bWareHouseCV14_Fwd                         : BIT; //Y7.0
        bWareHouseCV14_Rev                         : BIT; //Y7.1
        bWareHouseCV13_Fwd                         : BIT; //Y7.2
        bWareHouseCV13_Rev                         : BIT; //Y7.3
        bWareHouseCV12_Fwd                         : BIT; //Y7.4
        bWareHouseCV12_Rev                         : BIT; //Y7.5
        bWareHouseCV11_Fwd                         : BIT; //Y7.6
        bWareHouseCV11_Rev                         : BIT; //Y7.7
        bUpCV_Fwd                                  : BIT; //Y7.8
        bUpCV_Rev                                  : BIT; //Y7.9
        bLowCV_Fwd                                 : BIT; //Y7.10
        bLowCV_Rev                                 : BIT; //Y7.11
        bPullOutCV_A_Fwd                           : BIT; //Y7.12
        bPullOutCV_A_Rev                           : BIT; //Y7.13
        bPullOutCV_B_Fwd                           : BIT; //Y7.14
        bPullOutCV_B_Rev                           : BIT; //Y7.15
        bUpCV_DiameterHoriz_Extend_Valve           : BIT; //Y8.0
        bUpCV_DiameterHoriz_Retract_Valve          : BIT; //Y8.1
        bUpCV_DiameterVert_Valve                   : BIT; //Y8.2
        bUpCV_DiameterClamp_Close_Valve            : BIT; //Y8.3
        bUpCV_DiameterClamp_Open_Valve             : BIT; //Y8.4
        bStackPush_Valve                           : BIT; //Y8.5
        bCamara_Blow                               : BIT; //Y8.6
        Spare72                                    : BIT; //Y8.7
        bStorage_StartPbLamp                       : BIT; //Y8.8
        bStorage_StopPbLamp                        : BIT; //Y8.9
        bStorage_ResetPbLamp                       : BIT; //Y8.10
        bStorage_StackPushPbLamp                   : BIT; //Y8.11
        bStorage_EleBoxLight                       : BIT; //Y8.12
        bPullOutCV_FwdPbLamp                       : BIT; //Y8.13
        bPullOutCV_RevPbLamp                       : BIT; //Y8.14
        bStorage_FanucRobotPower                   : BIT; //Y8.15
        bStorage_SingleTower_BlueLamp              : BIT; //Y10.0
        bStorage_SingleTower_RedLamp           	   : BIT; //Y10.1
        bStorage_SingleTower_YellowLamp            : BIT; //Y10.2
        bStorage_SingleTower_GreenLamp             : BIT; //Y10.3
        bStorage_Buzzer                            : BIT; //Y10.4
        bTurnOffRS485Sensors_1                     : BIT; //Y10.5
        bTurnOffRS485Sensors_2                     : BIT; //Y10.6 // Customer request control RS485 module by Albert 20250910
        bStorage_AreaLight                         : BIT; //Y10.7
        bPullOutCV_AsidePress1_Valve               : BIT; //Y10.8
        bPullOutCV_AsidePress2_Valve               : BIT; //Y10.9
        bPullOutCV_AsideBlock_Valve                : BIT; //Y10.10
        bPullOutCV_BsidePress1_Valve               : BIT; //Y10.11
        bPullOutCV_BsidePress2_Valve               : BIT; //Y10.12
        bPullOutCV_BsideBlock_Valve                : BIT; //Y10.13
        Spare95                                    : BIT; //Y10.14
        Spare96                                    : BIT; //Y10.15
        bLowCV_Press1_Valve                        : BIT; //Y11.0
        bLowCV_Press2_Valve                        : BIT; //Y11.1
        bLowCV_Press3_Valve                        : BIT; //Y11.2
        bLowCV_Press4_Valve                        : BIT; //Y11.3
        bLowCV_Block1_Up_Valve                     : BIT; //Y11.4
        bLowCV_Block1_Down_Valve                   : BIT; //Y11.5
        bLowCV_Block2_Up_Valve                     : BIT; //Y11.6
        bLowCV_Block2_Down_Valve                   : BIT; //Y11.7
        Spare105                                   : BIT; //Y11.8
        Spare106                                   : BIT; //Y11.9
        bShippingTransCV_Leftside_Allow            : BIT; //Y11.10		// 我方給大族，左邊輸送帶的允許移動訊號
        Spare108                                   : BIT; //Y11.11
        bShippingTransCV_Rightside_Allow           : BIT; //Y11.12		// 我方給大族，右邊輸送帶的允許移動訊號
        Spare110                                   : BIT; //Y11.13
        Spare111                                   : BIT; //Y11.14
        Spare112                                   : BIT; //Y11.15
        bAllocateRobot_LeftVert1_Valve             : BIT; //Y0.0
        bAllocateRobot_LeftVert2_Valve             : BIT; //Y0.1
        bAllocateRobot_RightVert1_Valve            : BIT; //Y0.2
        bAllocateRobot_RightVert2_Valve            : BIT; //Y0.3
        bAllocateRobot_LeftClamp1_Close_Valve      : BIT; //Y0.4
        bAllocateRobot_LeftClamp1_Open_Valve       : BIT; //Y0.5
        bAllocateRobot_LeftClamp2_Close_Valve      : BIT; //Y0.6
        bAllocateRobot_LeftClamp2_Open_Valve       : BIT; //Y0.7
        bAllocateRobot_RightClamp1_Close_Valve     : BIT; //Y0.8
        bAllocateRobot_RightClamp1_Open_Valve      : BIT; //Y0.9
        bAllocateRobot_RightClamp2_Close_Valve     : BIT; //Y0.10
        bAllocateRobot_RightClamp2_Open_Valve      : BIT; //Y0.11
        bRoundBelt_WorkZone_Press_Valve            : BIT; //Y0.12
        bRoundBelt_WorkZone_Plug_Valve             : BIT; //Y0.13
        bRoundBelt_ChargeZone_Plug_Valve           : BIT; //Y0.14
        bRoundBelt_TransmitCVZone_Plug_Valve       : BIT; //Y0.15
        bOutRobot_AsideVert_Valve                  : BIT; //Y1.0
        bOutRobot_BsideVert_Valve                  : BIT; //Y1.1
        bOutRobot_AsideClamp_Close_Valve           : BIT; //Y1.2
        bOutRobot_AsideClamp_Open_Valve            : BIT; //Y1.3
        bOutRobot_BsideClamp_Close_Valve           : BIT; //Y1.4
        bOutRobot_BsideClamp_Open_Valve            : BIT; //Y1.5
        bTransmitCV_CamaraHorizDifferentSide_Valve  : BIT; //Y1.6
        bTransmitCV_CamaraHorizSameSizeSide_Valve: BIT; //Y1.7
        bDifferentSizeCV_Press2_Valve              : BIT; //Y1.8
        bDifferentSizeCV_Press1_Valve              : BIT; //Y1.9
        bDifferentSizeCV_Block1_Valve              : BIT; //Y1.10
        bSameSizeCV_Press4_Valve                   : BIT; //Y1.11
        bSameSizeCV_Press3_Valve                   : BIT; //Y1.12
        bSameSizeCV_Press2_Valve                   : BIT; //Y1.13
        bSameSizeCV_Press1_Valve                   : BIT; //Y1.14
        bSameSizeCV_Block2_Valve                   : BIT; //Y1.15
        bSameSizeCV_Block1_Valve                   : BIT; //Y2.0
        bTurntable_Press_Valve                     : BIT; //Y2.1
        bTransmitCV_SameSizeSide_Fwd               : BIT; //Y2.2
        bShipping_FanucRobotPower                  : BIT; //Y2.3
        bTransmitCV_DifferentSide_Fwd              : BIT; //Y2.4
        bTransmitCV_DifferentSide_Rev              : BIT; //Y2.5
        bAllocated_AreaLight                       : BIT; //Y2.6
        bTransmitCV_SameSide_Rev                   : BIT; //Y2.7
        bAllocated_SignalTower_RedLamp             : BIT; //Y2.8
        bAllocated_SignalTower_YellowLamp          : BIT; //Y2.9
        bAllocated_SignalTower_GreenLamp           : BIT; //Y2.10
        bAllocated_SignalTower_BlueLamp            : BIT; //Y2.11
        bAllocated_StartPbLamp                     : BIT; //Y2.12
        bAllocated_StopPbLamp                      : BIT; //Y2.13
        bAllocated_ResetPbLamp                     : BIT; //Y2.14
        bAllocated_Buzzer                          : BIT; //Y2.15

    END_STRUCT
END_TYPE

// ---- Library/10_Machine/19_Device/EL2889/ST_OutputTable_Mitsubishi.TcDUT
TYPE
    ST_OutputTable_Mitsubishi :
    STRUCT
        Y4  : uni_IntToBool;
        Y5  : uni_IntToBool;
        Y6  : uni_IntToBool;
        Y7  : uni_IntToBool;
        Y8  : uni_IntToBool;
        Y10 : uni_IntToBool;
        Y11 : uni_IntToBool;
        Y0  : uni_IntToBool;
        Y1  : uni_IntToBool;
        Y2  : uni_IntToBool;
    END_STRUCT
END_TYPE

// ---- Library/10_Machine/19_Device/EL2889/uni_OutputModule.TcDUT
TYPE
    uni_OutputModule :
    UNION
        stEbusDO : ST_EbusOutputModule;       // Output table defined based on module allocation.
        stDO     : ST_OutputTable;            // Output table defined based on variable names.
        stDIList : ST_OutputTable_Mitsubishi; // Output table defined based on Mitsubishi PLC convention.
    END_UNION
END_TYPE

// ---- Library/10_Machine/19_Device/FanucRobot/DUTs/ST_AutoMode_ShippingRobotTransfer.TcDUT
TYPE ST_AutoMode_ShippingRobotTransfer :
STRUCT
	Command          : ST_CommandBasic;
	Status           : ST_StatusBasic;
	Info             : ST_ShippingRobotTransfer_Info;
	bCompleteRequest : BOOL;              // buzz/lamp 完成警報觸發
	bTransCVInPosition_Left  : BOOL;    // 左側 TransCV sensor 到位狀態回饋
	bTransCVInPosition_Right : BOOL;    // 右側 TransCV sensor 到位狀態回饋
END_STRUCT
END_TYPE

// ---- Library/10_Machine/19_Device/FanucRobot/DUTs/ST_AutoMode_ShippingRobot_MoveAbs.TcDUT
TYPE ST_AutoMode_ShippingRobot_MoveAbs :
STRUCT
	Command 	: ST_CommandBasic;
	Status 		: ST_StatusBasic;
	Info 		: ST_RobotRegionMove_Info;
	bCompleteRequest 	: BOOL;
	bTransCVInPosition	: BOOL;
END_STRUCT
END_TYPE

// ---- Library/10_Machine/19_Device/FanucRobot/DUTs/ST_ReadWriteParaStatus.TcDUT
TYPE
    ST_ReadWriteParaStatus :
    STRUCT
        ReadCompleted  : BIT; // True : Read Offset data completed
        WriteCompleted : BIT; // True : Write Offset data completed
        Simulation     : BIT; // True : Fanuc robot some value to be force set
        AutoMode       : BIT; // True : Fanuc robot in Auto mode
        T1Mode         : BIT; // True : Fanuc robot in T1 mode, Manual mode in low speed.
        T2Mode         : BIT; // True : Fanuc robot in T2 mode, Manual mode in high speed.
        E_Stop         : BIT; // True : Fanuce robot teach pendant's Estop has be press.
        RSR1_Active    : BIT; // True : RSR1 prog is running
        RSR2_Active    : BIT; // True : RSR2 prog is running
        RSR3_Active    : BIT; // True : RSR3 prog is running
        BzoneInWork    : BIT; // True : Robot request to move in to allocate zone
        BzoneWaitAllow : BIT; //EzoneInWork    : BIT;
        JzoneInWork    : BIT;
		Space_1		   : BIT;	//======================Add Jidian Version V2 Robot ==================17~19 bit
		Space_2		   : BIT;
		A_Depot_Laser  : BIT; //ADepot Laser Status
    END_STRUCT
END_TYPE

// ---- Library/20_MachineUnits/21_StorageArea/Duts/E_FeedInToWareHouseAction.TcDUT
{attribute 'qualified_only'}
{attribute 'strict'}
TYPE E_FeedInToWareHouseAction :
(
	Undefined := 0,
	ClampA_WareHouseA,
	ClampA_WareHouseB,
	ClampB_WareHouseA,
	ClampB_WareHouseB,
	A_WareHouseA_B_WareHouseA,
	A_WareHouseA_B_WareHouseB,
	A_WareHouseB_B_WareHouseA,
	A_WareHouseB_B_WareHouseB
);
END_TYPE

// ---- Library/20_MachineUnits/21_StorageArea/Duts/st_RebootModbusDevices.TcDUT
TYPE st_RebootModbusDevices :
STRUCT
	Command 	: ST_CommandBasic;
	Status 		: ST_StatusBasic;
	OffDelayTime	: INT := 2; // Waitting time after power off in second		//default 2 s ,if C# no assign
	OnDelayTime		: INT; // Watting time after power on in second
END_STRUCT
END_TYPE

// ---- Library/20_MachineUnits/21_StorageArea/Duts/ST_StorageService.TcDUT
TYPE
    ST_StorageService :
    STRUCT
        // Automode Feedin empty box with robot 
        AutoMode_FeedInEmptyBoxWithRobot : REFERENCE TO ST_AutoMode_FeedInEmptyBox; // Automode : Feedin empty box with robot from Warehouse and Pullout convenyor
        // Automode Reload RoundBelt box with robot
        AutoMode_ReloadRoundBeltBoxWithRobot : REFERENCE TO ST_AutoMode_ReloadRoundBeltBox; // Automode : Reload RoundBelt box with robot from warehouse

		AutoMode_FeedInRoundBeltBoxToWareHouse : REFERENCE TO ST_AutoMode_FeedInToWareHouseBox;
        //AutoMode UpperFeedInConveyor
        AutoMode_UpperFeedInConveyor : REFERENCE TO ST_Auto_UpperFeedInConveyor;
        //AutoMode AddBoxes
        AutoMode_AddBoxes : REFERENCE TO ST_AutoAddsBoxes;

        //AutoModeUse------手臂區域移動_FeedIn conveyor
        AutoMode_RobotRegionMove_FeedInConveyor : REFERENCE TO ST_AutoMode_RobotRegionMove;
        //AutoModeUse------手臂區域移動_AllocatedConveyor
        AutoMode_RobotRegionMove_AllocatedConveyor : REFERENCE TO ST_AutoMode_RobotRegionMove;
        //AutoModeUse------手臂區域移動_Pullout conveyor
        AutoMode_RobotRegionMove_PullOutConveyor : REFERENCE TO ST_AutoMode_RobotRegionMove;
        //AutoModeUse------手臂區域移動_Buffer area
        AutoMode_RobotRegionMove_BufferArea : REFERENCE TO ST_AutoMode_RobotRegionMove;
        //AutoModeUse------手臂區域移動_RoundBelt
        AutoMode_RobotRegionMove_RoundBelt : REFERENCE TO ST_AutoMode_RobotRegionMove;

        // Pullout 
        AutoMode_PullOutConveyor : REFERENCE TO ST_AutoPullOutConveyor; // AutoMode PullOut Conveyor
        //AutoModeUse*-------手臂絕對位置移動
        AutoMode_RobotAbsMove : REFERENCE TO st_AutoSixAxisAbsMoveParameter;
        //        //AutoModeUse*-------手臂倉儲位置移動
        //        AutoMode_RobotWarehouseMove : st_AutoSixAxisWarehouseParameter;

        //AutoModeUse------倉儲馬達搭配手臂移動
        AutoMode_WarehouseMotoWithRobotMove : REFERENCE TO st_AutoSixAxisWarehouseParameter;
		
		//AutoModeUse------倉儲內取放圓帶 (單筆)
		AutoMode_WareHouseInnerPickToRoundBelt : REFERENCE TO ST_AutoMode_WareHouseInnerPickToRoundBelt;
		//AutoModeUse------倉儲內取放圓帶 (批次)
		AutoMode_WareHouseInnerPickToRoundBeltBatch : REFERENCE TO ST_WareHouseInnerPickBatch;
		//AutoModeUse------圓帶回倉/PullOut (批次)
		AutoMode_FeedInRoundBeltBoxBatch : REFERENCE TO ST_FeedInRBBatch;
		
		//Reboot Modbus devices
		RebootModbusDevices			: REFERENCE TO st_RebootModbusDevices;
		//AutoMode--------- 倉儲區六軸手臂單獨回原點
		AutoMode_RobotSelfHoming	: REFERENCE TO ST_AutoMode_RobotSelfHoming;
    END_STRUCT
END_TYPE

// ---- Library/20_MachineUnits/22_AllocateArea/Duts/ST_AllocateService.TcDUT
TYPE
    ST_AllocateService :
    STRUCT
        AllocateMoveStructure              : REFERENCE TO st_ads_AllocateMoveStructure;
        AllocateCircleMove                 : REFERENCE TO st_AllocateCircleMoveStructure;
        TurnTableMove                      : REFERENCE TO st_ads_OneAxisMoveWithPosition;
        AutoMode_AllocateBatchMode         : REFERENCE TO ST_AllocationJobBatchMode;
        AutoMode_SimpleAllocation_Batch    : REFERENCE TO ST_AllocationJobBatchMode;
        AutoMode_AllocateBatchMode_Reverse : REFERENCE TO ST_AllocationJobBatchMode;
        AutoMode_RareBoxMove               : REFERENCE TO st_AutoMode_ClampingBoxesJob;
        AutoMode_EmptyBoxMove              : REFERENCE TO st_AutoMode_ClampingBoxesJob;
        AutoMode_BoxMoveReverse            : REFERENCE TO st_AutoMode_ClampingBoxesJob;
        AutoMode_SameSizeCVCamera          : REFERENCE TO ST_AutoMode_TransCVCamera;
        AutoMode_SameSizeCVCamera_Reverse  : REFERENCE TO ST_AutoMode_TransCVCamera;
        AutoMode_DifferentCVCamera         : REFERENCE TO ST_AutoMode_TransCVCamera;
        AllocateRegionHome                 : REFERENCE TO st_RegionHome;
        AutoMode_PullOutConveyor           : REFERENCE TO ST_AutoPullOutConveyor;
		AutoMode_AllocateCircleMove 	   : REFERENCE TO st_AllocateCircleMoveStructure;
		AutoMode_TurnTableMove 			   : REFERENCE TO st_ads_OneAxisMoveWithPosition;
		AllocateRobotNeedlingMove 		   : REFERENCE TO st_AllocateRobotNeedlingMove;
		AutoMode_ReverseBatchPick		   : REFERENCE TO ST_AutoMode_ReverseBatchPick;
		AutoMode_ReverseBoxToWareHouse	   : REFERENCE TO ST_AutoMode_ReverseBoxToWareHouse;
    END_STRUCT
END_TYPE

// ---- Library/20_MachineUnits/22_AllocateArea/Duts/ST_AutoMode_ReverseBatchPick.TcDUT
TYPE ST_AutoMode_ReverseBatchPick :
STRUCT
	Command				: ST_CommandBasic;		// C# → PLC (Execute, Reset, Abort)
	Status				: ST_StatusBasic;		// PLC → C# (Done, Busy, Error)

	// ===== 鐵盤 Sensor (目前由 C# ADS 模擬寫入, 後續要改成獨立硬體訊號) =====
	bLeftPlateReady		: BOOL;				// 左鐵盤到位 sensor  // 後面要改成獨立硬體訊號
	bRightPlateReady	: BOOL;				// 右鐵盤到位 sensor  // 後面要改成獨立硬體訊號

	// ===== 鐵盤配置 (C# → PLC) =====
	LeftPlate			: ARRAY[0..3] OF BOOL;
	RightPlate			: ARRAY[0..3] OF BOOL;
	bLeftConfigReady	: BOOL;
	bRightConfigReady	: BOOL;

	// ===== 拍照 Handshake =====
	UseBoxCamera		: BOOL;				// PLC → C# (請求拍照)
	BoxCameraDone		: BOOL;				// C# → PLC (拍照完成)
	CameraIsOK			: BOOL;				// C# → PLC
	CameraWarehouse		: INT;				// C# → PLC (倉 1=A, 2=B)
	CameraLevel			: INT;				// C# → PLC (層 1~10)
	CameraTrack			: INT;				// C# → PLC (軌 1~20)

	// ===== 鐵盤狀態 (PLC → C#) =====
	bLeftPlateArrived	: BOOL;
	bRightPlateArrived	: BOOL;
	bLeftPlateDone		: BOOL;
	bRightPlateDone		: BOOL;

	// ===== 狀態監控 (PLC → C#) =====
	uiUnphotographedCount	: UINT;
	uiTotalProcessed		: UINT;
	uiTransportedCount		: UINT;
END_STRUCT
END_TYPE

// ---- Library/20_MachineUnits/22_AllocateArea/Duts/E_ReverseBoxDestination.TcDUT
{attribute 'qualified_only'}
{attribute 'strict'}
(* 同尺寸軌道逆向送盒目的地
   WareHouse  : 入倉 (走 WareHouse.M_StartFeedInBox + StorageRobot.M_StartWareHousePlaceBox)
   PullOut    : 回拔輸送帶 (走 FB_RobotRegionMove_PullOutConveyor)
   NGConveyor : 倉儲區軌道 NG 位置 (E_RobotArea.InOutConveyor Position 3,走 FB_RobotRegionMove_FeedInConveyor_V2)
*)
TYPE E_ReverseBoxDestination :
(
	WareHouse	:= 0,
	PullOut		:= 1,
	NGConveyor	:= 2
);
END_TYPE

// ---- Library/20_MachineUnits/22_AllocateArea/Duts/ST_AutoMode_ReverseBoxToWareHouse.TcDUT
// ST_AutoMode_ReverseBoxToWareHouse
// 逆向拍照批次 — 大手臂搬運入倉 / PullOut / NG 的 ADS Handshake 結構
// C# HMI 透過 ADS 讀寫此結構，對應 FB_SameSizeCV_ReverseBoxToWareHouse
// 支援: 單爪A / 單爪B / 雙爪 (A+B 兩盒連續搬運)
//
// 介面變更 (2026-05-13): bBoxA/B_IsOK BOOL 改成 eBoxA/B_Destination enum,新增 PullOut 目的地
TYPE ST_AutoMode_ReverseBoxToWareHouse :
STRUCT
	Command		: ST_CommandBasic;		// [ADS Write] C# → PLC : Execute=啟動, Reset=復位, Abort=中止
	Status		: ST_StatusBasic;		// [ADS Read]  PLC → C# : Done=完成, Busy=執行中, Error=異常

	// ===== A爪 盒子資訊 (C# → PLC, ADS Write) =====
	bBoxA_Enable		: BOOL;						// TRUE=A爪有盒子要處理, FALSE=不使用A爪
	eBoxA_Destination	: E_ReverseBoxDestination;	// A爪目的地: WareHouse / PullOut / NGConveyor
	iBoxA_Warehouse		: INT;						// (僅 Destination=WareHouse) 目標倉別 E_WareHouse: 1=A, 2=B
	iBoxA_Level			: INT;						// (僅 Destination=WareHouse) 目標層 1~10
	iBoxA_Track			: INT;						// (僅 Destination=WareHouse) 目標軌 1~20
	iBoxA_PullOutSide	: INT;						// (僅 Destination=PullOut) 1=I3_Slide 左 / 2=I4_Slide 右

	// ===== B爪 盒子資訊 (C# → PLC, ADS Write) =====
	bBoxB_Enable		: BOOL;						// TRUE=B爪有盒子要處理, FALSE=不使用B爪 (單爪模式)
	eBoxB_Destination	: E_ReverseBoxDestination;
	iBoxB_Warehouse		: INT;
	iBoxB_Level			: INT;
	iBoxB_Track			: INT;
	iBoxB_PullOutSide	: INT;						// 1=I3_Slide 左 / 2=I4_Slide 右

	// ===== 狀態回饋 (PLC → C#, ADS Read) =====
	bBoxA_Done			: BOOL;						// A爪搬運完成 (入倉/PullOut/NG 三路皆算完成)
	bBoxB_Done			: BOOL;						// B爪搬運完成
END_STRUCT
END_TYPE

// ---- Library/20_MachineUnits/22_AllocateArea/Duts/ST_ReverseBatchBoxQueue.TcDUT
TYPE ST_ReverseBatchBoxQueue :
STRUCT
	Boxes		: ARRAY[0..15] OF ST_ReverseBatchBoxResult;	// 環形佇列
	WriteIdx	: UINT;		// FB_A 寫入位置
	ReadIdx		: UINT;		// 大手臂讀取位置
	Count		: UINT;		// 待搬運數量
END_STRUCT
END_TYPE

// ---- Library/20_MachineUnits/22_AllocateArea/Duts/ST_ReverseBatchBoxResult.TcDUT
TYPE ST_ReverseBatchBoxResult :
STRUCT
	bActive		: BOOL;		// 此 slot 有資料
	bIsOK		: BOOL;		// 拍照結果 OK/NG
	iWarehouse	: INT;		// 倉 (OK 時有效)
	iLevel		: INT;		// 層 (OK 時有效)
	iTrack		: INT;		// 軌 (OK 時有效)
END_STRUCT
END_TYPE

// ---- Library/20_MachineUnits/23_ShippingArea/Duts/ST_BlinkInfo.TcDUT
TYPE ST_BlinkInfo :
STRUCT
	BuzzCount		: UINT;
	LightCount		: UINT;	
	MaxBuzzCOunt    : UINT := 3;
	MaxLightCount	: UINT := 3;
	trigBizz		:R_TRIG;
	TrigLight		:R_TRIG;
END_STRUCT
END_TYPE

// ---- Library/20_MachineUnits/23_ShippingArea/Duts/ST_ShippingRobotTransfer_AreaInfo.TcDUT
TYPE ST_ShippingRobotTransfer_AreaInfo :
STRUCT
	Area     : E_RobotArea;   // 目標區域 (8=Left, 9=Right, 10=TransmitCVEnd, 11=Buffer, 12=CCD)
	Position : INT;           // 位置地址 (0=CCD, 1-55=Buffer, 1-2=TransmitCVEnd, 1-40=Left/Right)
	Get      : BOOL;          // TRUE=取盒, FALSE=放盒
END_STRUCT
END_TYPE

// ---- Library/20_MachineUnits/23_ShippingArea/Duts/ST_ShippingRobotTransfer_Info.TcDUT
TYPE ST_ShippingRobotTransfer_Info :
STRUCT
	Source      : ST_ShippingRobotTransfer_AreaInfo;   // 來源
	Destination : ST_ShippingRobotTransfer_AreaInfo;   // 目標
END_STRUCT
END_TYPE

// ---- Library/20_MachineUnits/23_ShippingArea/Duts/ST_ShippingService.TcDUT
TYPE
    ST_ShippingService :
    STRUCT
        AutoMode_ShippingRobot_Left          : REFERENCE TO ST_AutoMode_ShippingRobot_MoveAbs;
        AutoMode_ShippingRobot_Right         : REFERENCE TO ST_AutoMode_ShippingRobot_MoveAbs;
        AutoMode_ShippingRobot_TransmitCVEnd : REFERENCE TO ST_AutoMode_ShippingRobot_MoveAbs;
		AutoMode_ShippingTransCV_LeftSide	 : REFERENCE TO ST_AutoMode_ShippingLeftSideTransCV;
		AutoMode_ShippingTransCV_RightSide	 : REFERENCE TO ST_AutoMode_ShippingRightSideTransCV;
		AutoMode_ShippingRobot_Buffer		 	: REFERENCE TO ST_AutoMode_ShippingRobot_MoveAbs;
		AutoMode_ShippingRobot_PhotoStandByPos	: REFERENCE TO ST_AutoMode_ShippingRobot_MoveAbs;
		AutoMode_ShippingRobotTransfer			: REFERENCE TO ST_AutoMode_ShippingRobotTransfer;
		AutoMode_ShippingPlateScan				: REFERENCE TO ST_ShippingPlateToConveyor;
    END_STRUCT
END_TYPE

// ---- POUs/RS485_JidianVersion/DUTs/ST_RS485Controller.TcDUT
TYPE ST_RS485Controller :
STRUCT
	stSliderStatusALL:ST_RS485_SliderStatusALL;
	stLayerStatus:ST_RS485_LayerStatus;
	stHeartbeat:ST_RS485_Heartbeat;	
END_STRUCT
END_TYPE

// ---- POUs/RS485_JidianVersion/DUTs/ST_RS485_Heartbeat.TcDUT
TYPE ST_RS485_Heartbeat :
STRUCT
	nHeartbeat1:BIT;
	nHeartbeat2:BIT;
	nHeartbeat3:BIT;
	nHeartbeat4:BIT;
	nHeartbeat5:BIT;
	nHeartbeat6:BIT;
	nHeartbeat7:BIT;
	nHeartbeat8:BIT;
	nHeartbeat9:BIT;
	nHeartbeat10:BIT;	
END_STRUCT
END_TYPE

// ---- POUs/RS485_JidianVersion/DUTs/ST_RS485_LayerStatus.TcDUT
TYPE ST_RS485_LayerStatus :
STRUCT
	nPCB1:BIT;
	nPCB2:BIT;
	nPCB3:BIT;
	nPCB4:BIT;
	nPCB5:BIT;
	nPCB6:BIT;
	nPCB7:BIT;
	nPCB8:BIT;
	nPCB9:BIT;
	nPCB10:BIT;
END_STRUCT
END_TYPE

// ---- POUs/RS485_JidianVersion/DUTs/ST_RS485_SliderStatusALL.TcDUT
TYPE ST_RS485_SliderStatusALL :
STRUCT
	bPos:ARRAY[1..100]OF BOOL;
END_STRUCT
END_TYPE

// ---- Library/10_Machine/12_MachineControl/GVL_Machine.TcGVL
VAR_GLOBAL
    PackTags               : ARRAY[0..3] OF ST_PackMLv30; //PackTags
    bButtonProductionReq   : BOOL; //TRUE when a mode change to PRODUCTION is requested
    stChangeIntoProduction : ST_ChangeIntoProduction; //Result of command box "Change to Production requested"
    CylinderStatus         : ST_CylinderStatus;
    RemoteData             : ST_SetupPara;
    AllocatYAxisHome       : BOOL;
	stModbusByPassInternal : st_ModbusSwitchOff;

END_VAR
VAR_GLOBAL PERSISTENT
    LocalData : ST_SetupPara;
END_VAR

// ---- Library/10_Machine/12_MachineControl/GVL_Machine_Const.TcGVL
VAR_GLOBAL CONSTANT
	udiMax_CylinderNum : UDINT := 54;
END_VAR

// ---- Library/10_Machine/13_ErrorHandling/GVL_ErrorCode.TcGVL

(*
=================================================================================
    全域錯誤碼定義

    [1] GC_ALARM_xxx — RegisterAlarm ID (DINT)，FB_MachineControl 使用，HMI 顯示
    [2] GC_ERR_xxx   — FB 內部錯誤碼 (INT, AOOEE 編碼)，各 FB M_GetErrorMsg 使用

    續作標記: [Hold]=暫停可恢復, [Abort]=必須停機
    擴充原則: 每區段保留 50%+ 空位，新增從尾端往後排
=================================================================================
*)
{attribute 'qualified_only'}
VAR_GLOBAL CONSTANT

    // =========================================================================
    // [1] RegisterAlarm ID — Homing 服務 (10-99)
    // =========================================================================
    GC_ALARM_MACHINE_HOMING              : DINT := 10;    // [Hold] 機台回原點錯誤
    GC_ALARM_STORAGE_HOMING              : DINT := 11;    // [Hold] 倉儲區回原點錯誤
    GC_ALARM_ALLOCATE_HOMING             : DINT := 12;    // [Hold] 配針區回原點錯誤
    GC_ALARM_SHIPPING_HOMING             : DINT := 13;    // [Hold] 出貨區回原點錯誤
    GC_ALARM_TABLE_MOVE                  : DINT := 14;    // [Hold] TableMove 錯誤
    GC_ALARM_MODBUS_RTU                  : DINT := 15;    // [Hold] Modbus RTU 通訊
    GC_ALARM_MACHINEMODE_SWITCH          : DINT := 16;    // [Hold] 機台模式切換
    // 16-99: 預留 Homing/通用服務擴充

    // =========================================================================
    // [1] RegisterAlarm ID — 倉儲區服務 (100-199)
    // =========================================================================
    GC_ALARM_STO_RELOAD_BOX              : DINT := 100;   // [Hold] 補盒服務
    GC_ALARM_STO_FEEDIN_BOX              : DINT := 101;   // [Hold] 進盒服務
    GC_ALARM_STO_ADD_BOXES               : DINT := 102;   // [Hold] 加盒服務
    GC_ALARM_STO_BOX_SUPPLY              : DINT := 103;   // [Hold] 供盒控制
    GC_ALARM_STO_FEEDIN_EMPTY            : DINT := 104;   // [Hold] 空盒入倉
    GC_ALARM_STO_RELOAD_ROUNDBELT        : DINT := 105;   // [Hold] 圓帶補盒
    GC_ALARM_STO_ROBOT_ABS_MOVE          : DINT := 106;   // [Hold] 機器人絕對移動
    GC_ALARM_STO_REGION_ALLOC_CV         : DINT := 107;   // [Hold] 區域移動-配針輸送帶
    GC_ALARM_STO_REGION_BUFFER           : DINT := 108;   // [Hold] 區域移動-緩衝區
    GC_ALARM_STO_REGION_FEEDIN_CV        : DINT := 109;   // [Hold] 區域移動-進料輸送帶
    GC_ALARM_STO_REGION_PULLOUT_CV       : DINT := 110;   // [Hold] 區域移動-拔針輸送帶
    GC_ALARM_STO_REGION_ROUNDBELT        : DINT := 111;   // [Hold] 區域移動-圓帶
    GC_ALARM_STO_UPPER_FEEDIN_CV         : DINT := 112;   // [Hold] 上層進料輸送帶
    GC_ALARM_STO_WAREHOUSE_ROBOT         : DINT := 113;   // [Hold] 倉儲機器人移動
    GC_ALARM_STO_CABINET_FEEDIN          : DINT := 114;   // [Hold] 料櫃進盒
    GC_ALARM_STO_CABINET_RELOAD          : DINT := 115;   // [Hold] 料櫃補盒
    GC_ALARM_STO_FEEDIN_RB_TO_WH         : DINT := 116;   // [Hold] 圓帶盒入倉
    GC_ALARM_STO_DIAMETER_MOVEMENT       : DINT := 117;   // [Hold] 直徑移動
	GC_ALARM_STO_ROBOTSELFHOMING		 : DINT := 118;	  // [Hold] 倉儲區手臂單獨回原點
	GC_AlARM_STO_ROBOTINNERPICK			 : DINT := 119;	  // [Hold] 倉儲分揀放置圓帶
	GC_AlARM_STO_ROBOTINNERPICK_BATCH	 : DINT := 120;	  // [Hold] 倉儲分揀放置圓帶BATCH
	GC_AlARM_STO_ROUNDBELTTOWAREHOUSE_BATCH	 : DINT := 121;	  // [Hold] 圓帶回倉ATCH

    // 119-199: 預留倉儲區服務擴充

    // =========================================================================
    // [1] RegisterAlarm ID — 配針區服務 (200-299)
    // =========================================================================
      GC_ALARM_ALC_BATCH_MODE              	: DINT := 200;   // [Hold] 批次配針
    GC_ALARM_ALC_BATCH_REVERSE           	: DINT := 201;   // [Hold] 批次配針反向
    GC_ALARM_ALC_DIFF_CV_CAMERA          	: DINT := 202;   // [Hold] 異徑CV相機
    GC_ALARM_ALC_OUTROBOT_REVERSE        	: DINT := 203;   // [Hold] OutRobot 反向移盒
    GC_ALARM_ALC_OUTROBOT_EMPTY          	: DINT := 204;   // [Hold] OutRobot 空盒移動
    GC_ALARM_ALC_OUTROBOT_RARE           	: DINT := 205;   // [Hold] OutRobot 稀有盒移動
    GC_ALARM_ALC_PULLOUT_CV              	: DINT := 206;   // [Hold] 拔針輸送帶
    GC_ALARM_ALC_ROUNDBELT               	: DINT := 207;   // [Hold] 圓帶控制
    GC_ALARM_ALC_SAME_CV_CAMERA          	: DINT := 208;   // [Hold] 同徑CV相機
    GC_ALARM_ALC_TURNTABLE               	: DINT := 209;   // [Hold] 轉盤控制
    GC_ALARM_ALC_OUTROBOT_TT_TO_RB       	: DINT := 210;   // [Hold] OutRobot 轉盤→圓帶
    GC_ALARM_ALC_NEEDLING_MOVE           	: DINT := 211;   // [Hold] 配針移動
    GC_ALARM_ALC_SAME_CV_CAMERA_REVERSE  	: DINT := 212;   // [Hold] 同徑CV相機(反向)
	GC_ALARM_ALC_REVERSE_TO_WAREHOUSE       : DINT := 213;   // [Hold] 反轉輸送帶入倉
	GC_ALARM_ALC_REVERSE_TO_WAREHOUSE_BATCH : DINT := 214;   // [Hold] 反轉輸送帶入倉Batch
	
    // 212-299: 預留配針區服務擴充

    // =========================================================================
    // [1] RegisterAlarm ID — 出貨區服務 (300-399)
    // =========================================================================
    GC_ALARM_SHP_ROBOT_LEFT              : DINT := 300;   // [Hold] 出貨機器人左
    GC_ALARM_SHP_ROBOT_RIGHT             : DINT := 301;   // [Hold] 出貨機器人右
    GC_ALARM_SHP_ROBOT_TRANSMIT_END      : DINT := 302;   // [Hold] 出貨機器人傳送端
    GC_ALARM_SHP_LEFT_TRANS_CV           : DINT := 303;   // [Hold] 左側傳送帶
    GC_ALARM_SHP_RIGHT_TRANS_CV          : DINT := 304;   // [Hold] 右側傳送帶
    GC_ALARM_SHP_ROBOT_BUFFER            : DINT := 305;   // [Hold] 出貨機器人緩衝
    GC_ALARM_SHP_ROBOT_TRANSFER          : DINT := 306;   // [Hold] 出貨機器人轉移
	GC_ALARM_SHP_ROBOT_PHOTOSTANDBYPOS   : DINT := 307;   // [Hold] 出貨機器人拍照等待位
	GC_ALARM_SHP_ROBOT_SCANPICK		     : DINT := 308;   // [Hold] 出貨機器人大族輸送帶掃描取盒

    // 307-399: 預留出貨區服務擴充

